# B&R Automation Studio project Lab2_Conveyor (part 3)

#### StateMoveToMagazine.ld
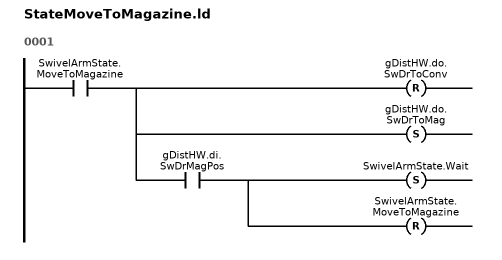
Ladder, written as Structured Text:
```iecst
ACTION StateMoveToMagazine:
VAR
    _p1 : BOOL;
END_VAR
(* Network 1 *)
IF SwivelArmState.MoveToMagazine THEN
    gDistHW.do.SwDrToConv := FALSE;
    gDistHW.do.SwDrToMag := TRUE;
END_IF;
_p1 := SwivelArmState.MoveToMagazine AND gDistHW.di.SwDrMagPos;
IF _p1 THEN
    SwivelArmState.Wait := TRUE;
    SwivelArmState.MoveToMagazine := FALSE;
END_IF;
END_ACTION
```

### Program Logical/Distributing/AlarmCtrl (IEC) - Alarm control for distributor

#### Cyclic.ld - Cyclic code
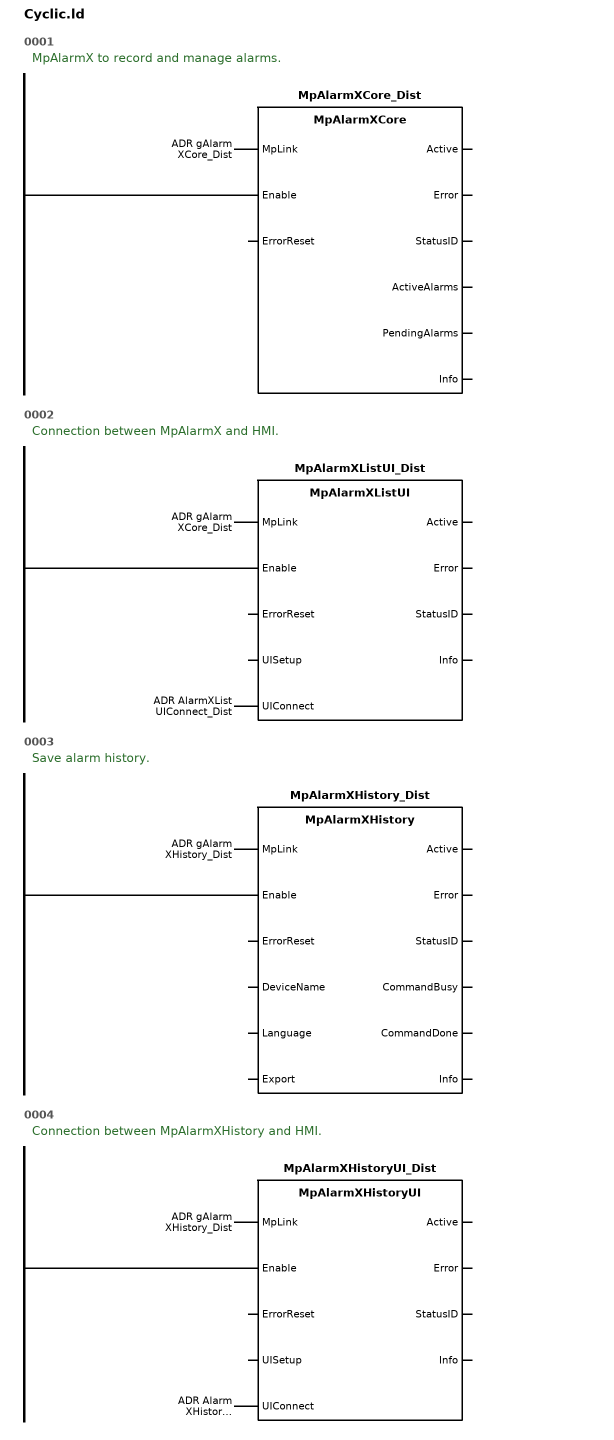
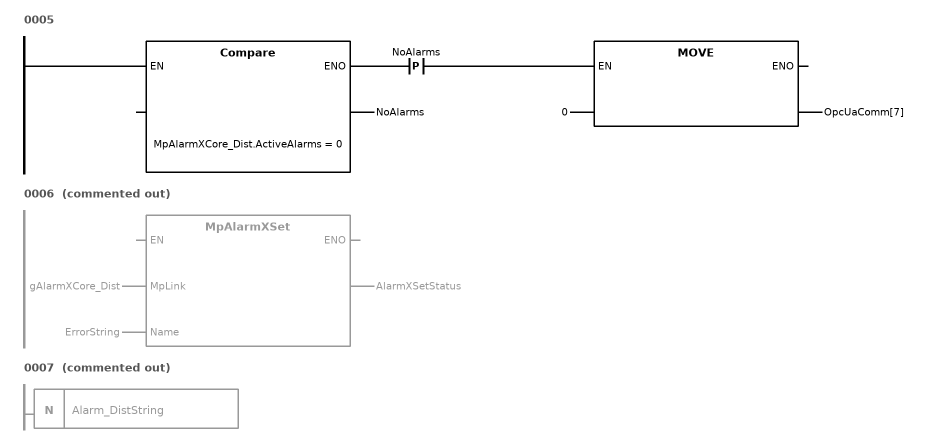
Ladder, written as Structured Text:
```iecst
(*********************************************************************************
 * Copyright: 	Hartfiel Automation
 * Author:    	cashley
 * Created:   	March 8, 2019/12:40 PM
 * Description: 	This file contains alarm handling for the distributing 			station.
 *********************************************************************************)
PROGRAM _CYCLIC
VAR
    _e1 : R_TRIG;
END_VAR
(* Network 1: MpAlarmX to record and manage alarms. *)
MpAlarmXCore_Dist(MpLink := ADR(gAlarmXCore_Dist), Enable := TRUE);

(* Network 2: Connection between MpAlarmX and HMI. *)
MpAlarmXListUI_Dist(MpLink := ADR(gAlarmXCore_Dist), Enable := TRUE, UIConnect := ADR(AlarmXListUIConnect_Dist));

(* Network 3: Save alarm history. *)
MpAlarmXHistory_Dist(MpLink := ADR(gAlarmXHistory_Dist), Enable := TRUE);

(* Network 4: Connection between MpAlarmXHistory and HMI. *)
MpAlarmXHistoryUI_Dist(MpLink := ADR(gAlarmXHistory_Dist), Enable := TRUE, UIConnect := ADR(AlarmXHistoryUIConnect_Dist));

(* Network 5 *)
NoAlarms := MpAlarmXCore_Dist.ActiveAlarms = 0;
_e1(CLK := NoAlarms);
IF _e1.Q THEN OpcUaComm[7] := 0; END_IF;

(* Network 6 *) (* commented out *)
// AlarmXSetStatus := MpAlarmXSet(MpLink := gAlarmXCore_Dist, Name := ErrorString);

(* Network 7 *) (* commented out *)
// Alarm_DistString;
END_PROGRAM
```

#### Variables.var - Local variables
```iecst
VAR
	MpAlarmXCore_Dist : MpAlarmXCore; (*Funciton block for MpAlarmXCore*)
	MpAlarmXListUI_Dist : MpAlarmXListUI; (*Function block for MpAlarmXListUI*)
	AlarmXListUIConnect_Dist : MpAlarmXListUIConnectType; (*MpAlarmXListUIConnect type*)
	MpAlarmXHistory_Dist : MpAlarmXHistory; (*Function block for MpAlarmXHistory*)
	MpAlarmXHistoryUI_Dist : MpAlarmXHistoryUI; (*Function block for MpAlarmXHistoryUI*)
	AlarmXHistoryUIConnect_Dist : MpAlarmXHistoryUIConnectType; (*MpAlarmXHistoryUIConnect type*)
	ErrorString : STRING[255]; (*String for MpAlarmXSet*)
	AlarmXSetStatus : UDINT; (*Output status for AlarmXSet*)
	NoAlarms : BOOL;
END_VAR
```

#### Alarm_DistString.st - Alarm action file
```iecst
ACTION Alarm_DistString:

END_ACTION
```

### DistMain.typ - Package global types
```iecst
TYPE
	AutoManualSelector_Enum :
		( (*Enumeration of manual-automatic mode*)
		DISTCTRL_AUTO := 0,
		DISTCTRL_MANUAL := 1
		);
	MainCtrlRejectionCode_Enum :
		( (*Enumeration of rejection codes thrown in response to a user requesting an illegal manual action.*)
		DIST_IN_AUTO_MODE := 0, (*Rejection Code thrown when any manual command is issued while the machine is in automatic mode.*)
		EJECTOR_EXTEND_PUCK_IN_TRAY := 1, (*Rejection Code thrown when an ejector extension is requested with a puck already in the ejector tray.*)
		EJECTOR_EXTEND_SWIVEL_IN_TRAY := 2, (*Rejection Code thrown when an ejector is requested with the swivel arm in the magazine position.*)
		SWIVEL_MOVE_MAG_HOLDING_PUCK := 3, (*Rejection Code thrown when the user tries to move the swivel arm to the magazine while the arm is holding a puck. Prevents pucks from being moved back to the ejector station, once removed.*)
		SWIVEL_MOVE_CONV_PUCK_CONFLICT := 4, (*Rejection Code thrown when the user attempts to transfer a puck to the conveyor with a puck already at the conveyor start position.*)
		SWIVEL_VAC_ON_NO_PRODUCT := 5, (*Rejection Code thrown when the user attempts to activate the swivel arm vacuum when there is no product under the suction cup.*)
		SWIVEL_VAC_OFF_PUCK_IN_TRANSIT := 6, (*Rejection Code thrown when the user attempts to deactivate the swivel arm vacuum while a puck is held and the swivel arm is in an intermediate position.*)
		CONV_JOG_BACK_PUCK_AT_START := 7, (*Rejection Code thrown when the user attempts to jog the conveyor backwards such that a puck falls off the conveyor.*)
		DIST_REJECT_PLACEHOLDER := 999,
		EJECTOR_EXTEND_ALREADY_IN_POS := 8, (*Rejection Code thrown when the user attempts to extend the ejection cylinder when it is already in the extended position.*)
		EJECTOR_RETRACT_ALREADY_IN_POS := 9, (*Rejection Code thrown when the user attempts to retract the ejection cylinder when it is already in the retracted position.*)
		SWIVEL_TO_MAG_ALREADY_IN_POS := 10, (*Rejection Code thrown when the user attempts to move the Swivel Arm to the magazine while to Swivel arm is already in that position.*)
		SWIVEL_TO_CONV_ALREADY_IN_POS := 11 (*Rejection Code thrown when the user attempts to move the Swivel Arm to the conveyor while to Swivel arm is already in that position.*)
		);
	MainCtrl_typ : 	STRUCT  (*Top-level interface structure for the MainCtrl task*)
		Input : MainCtrlInput_typ;
		Output : MainCtrlOutput_typ;
	END_STRUCT;
	MainCtrlInput_typ : 	STRUCT  (*Contains command and parameter substructures for the MainCtrl interface*)
		Cmd : MainCtrlCmd_typ; (*Command for MainCtrl*)
		Par : MainCtrlPar_typ; (*Parameters for MainCtrl*)
	END_STRUCT;
	MainCtrlCmd_typ : 	STRUCT  (*Contains commands for the MainCtrl interface*)
		StartAuto : BOOL;
		StopAuto : BOOL;
		Home : BOOL;
		Ejector : MainCtrlCmdEjector_typ; (*Contains a command substructure for the Ejector station*)
		SwivelArm : MainCtrlCmdSwivelArm_typ; (*Contains a command substructure for the Swivel Arm station*)
		Conveyor : MainCtrlCmdConveyor_typ; (*Contains a command substructure for the Conveyor station*)
		Reset : BOOL;
	END_STRUCT;
	MainCtrlCmdEjector_typ : 	STRUCT  (*Contains commands for the Ejector station*)
		Extend : BOOL; (*Command to extend the Ejector cylinder*)
		Retract : BOOL; (*Command to retract the Ejector cylinder*)
	END_STRUCT;
	MainCtrlCmdSwivelArm_typ : 	STRUCT  (*Contains commands for the Swivel Arm station*)
		MoveToConveyor : BOOL; (*Command to move the Swivel Arm to the Conveyor position*)
		MoveToMagazine : BOOL; (*Command to move the Swivel Arm to the magazine (i.e. Ejector) position*)
		VacuumOnImpulse : BOOL; (*Command to activate the Swivel Arm vacuum for an impulse. Used to pick up products.*)
		VacuumOffImpulse : BOOL; (*Command to active the Swivel Arm vacuum ejection impulse. Used to drop products.*)
	END_STRUCT;
	MainCtrlCmdConveyor_typ : 	STRUCT  (*Contains commands for the Conveyor station*)
		JogFwd : BOOL; (*Command to jog the Conveyor forward.*)
		JogBack : BOOL; (*Command to jog the Conveyor backward.*)
	END_STRUCT;
	MainCtrlPar_typ : 	STRUCT  (*Contains parameters for the MainCtrl task*)
		Mode : AutoManualSelector_Enum; (*Parameter to select manual/automatic operation.*)
		Conveyor : MainCtrlParConveyor_typ; (*Contains parameters for the Conveyor station*)
	END_STRUCT;
	MainCtrlParConveyor_typ : 	STRUCT  (*Contains parameters for the Conveyor station*)
		Speed : REAL; (*Parameter to set the speed of the conveyor. This value is applied to the Jog Forward, Jog Backward, and MoveVelocity actions for the conveyor.*)
		Accel : REAL; (*Parameter to set the acceleration of the conveyor. This value is applied to the Jog Forward, Jog Backward, and MoveVelocity actions for the conveyor.*)
		Decel : REAL; (*Parameter to set the deceleration of the conveyor. This value is applied to the Jog Forward, Jog Backward, and MoveVelocity actions for the conveyor.*)
	END_STRUCT;
	MainCtrlOutput_typ : 	STRUCT  (*Contains Status and "Command Rejected" information related to the MainCtrl task*)
		CommandRejected : BOOL; (*Output to indicate that a requested command is not allowed at a given time. True if the command is forbidden, false otherwise.*)
		RejectionCode : MainCtrlRejectionCode_Enum; (*Provides more detailed information about which command was rejected, and why.*)
		Status : MainCtrlStatus_typ; (*Provides additional status information about the MainCtrl task.*)
	END_STRUCT;
	MainCtrlStatus_typ : 	STRUCT  (*Contains status information about the MainCtrl task*)
		AutoRunTime : TIME; (*Time the machine has continuously been in automatic mode.*)
		DistProductCount : UDINT; (*Counter for how many products have been distributed by the distribution side of the machine.*)
		IsHomed : BOOL; (*Indicates whether the distribution half of the machine has been homed. True of the machine is homed.*)
	END_STRUCT;
END_TYPE
```

### DistMain.var - Package global variables
```iecst
VAR
	OpcUaComm : ARRAY[0..7] OF USINT; (*Communcation structure for OPCUA*)
	MainCtrl : MainCtrl_typ := (Input:=(Par:=(Mode:=DISTCTRL_MANUAL,Conveyor:=(Speed:=15.0,Accel:=200.0,Decel:=200.0)))); (*MainCtrl interface structure*)
END_VAR
```

### Program Logical/Distributing/dummyprog

#### Variables.var
```iecst
VAR
	ButtonLocked : ARRAY[0..2,0..2] OF BOOL := [FALSE,2(TRUE),FALSE,2(TRUE),FALSE,2(TRUE)];
	ButtonPressed : ARRAY[0..2,0..2] OF BOOL := [TRUE,2(FALSE),TRUE,2(FALSE),TRUE,2(FALSE)];
	i : USINT := 0;
	colourassigned : BOOL := FALSE;
	Lane : USINT := 0;
	Colour : USINT := 0;
END_VAR
VAR CONSTANT
	NUMBER_OF_LANES : USINT := 3;
	NUMBER_OF_COLOURS : USINT := 3;
	MAI_LANES : USINT := NUMBER_OF_LANES - 1;
	MAI_COLOURS : USINT := NUMBER_OF_COLOURS - 1;
END_VAR
VAR
	RTRIG : ARRAY[0..2,0..2] OF R_TRIG;
END_VAR
```

#### Cyclic.st
```iecst
PROGRAM _CYCLIC
	FOR Colour := 0 TO MAI_COLOURS BY 1 DO
		FOR Lane := 0 TO MAI_LANES BY 1 DO
			RTRIG[Colour,Lane].CLK := ButtonPressed[Colour,Lane];
		END_FOR
	END_FOR

	FOR Colour := 0 TO MAI_COLOURS BY 1 DO
		colourassigned := FALSE;
		FOR Lane := 0 TO MAI_LANES BY 1 DO
			IF ButtonPressed[Colour,Lane] THEN
				colourassigned := TRUE;
				FOR i := 0 TO MAI_LANES BY 1 DO
					IF i <> Lane THEN
						ButtonLocked[Colour,i] := TRUE;
					END_IF
				END_FOR
			END_IF
		END_FOR

		IF colourassigned = FALSE THEN
			FOR Lane := 0 TO MAI_LANES BY 1 DO
				ButtonLocked[Colour,Lane] := FALSE;
			END_FOR
		END_IF
	END_FOR

	FOR Lane := 0 TO MAI_LANES BY 1 DO
		FOR Colour := 0 TO MAI_COLOURS BY 1 DO
			IF RTRIG[Colour,Lane].Q THEN
				FOR i := 0 TO MAI_COLOURS BY 1 DO
					ButtonPressed[i,Lane] := FALSE;
				END_FOR
			END_IF
		END_FOR
	END_FOR

	FOR Colour := 0 TO MAI_COLOURS BY 1 DO
		FOR Lane := 0 TO MAI_LANES BY 1 DO
			RTRIG[Colour,Lane]();
		END_FOR
	END_FOR

END_PROGRAM
```

### Package Logical/Sorting - Sorter configuration

### Package Logical/Sorting/gAxisSortobj - gAxisSortobj

### Data object Logical/Sorting/gAxisSortobj/gAxisSorta (Apt) - gAxisSorta

#### gAxisSorta.apt
```
AcoposParameterTable:
  Root Parameters:
    64232 = 51200 (Name=SM_SCALE_STEP)
    64233 = 1000 (Name=SM_SCALE_LOAD_UNITS)
    64234 = 1 (Name=SM_SCALE_LOAD_MOTREV)
    230 = PCTRL_S_SET (Name=PCTRL_S_ACT_PARID)  // CTRL Position controller: Actual encoder position parameter ID
```

- Data object Logical/Sorting/gAxisSortobj/gAxisSorti (Ax) - gAxisSorti (no source held here)

### SortGlobal.var - Package global variables
```iecst
VAR
	gSortHW : gSortHW_type; (*Control variable for hardware IO types for sorter*)
	MpAlarmXCore_Sort : MpAlarmXCore; (*Function block for MpAlarmXCore*)
	MpAlarmXListUI_Sort : MpAlarmXListUI; (*Function block for MpAlarmXListUI*)
	AlarmXListUIConnect_Sort : MpAlarmXListUIConnectType; (*MpAlarmXListUIConnect type*)
	MpAlarmXHistory_Sort : MpAlarmXHistory; (*Function block for MpAlarmXHistory*)
	MpAlarmXHistoryUI_Sort : MpAlarmXHistoryUI; (*Function block for MpAlarmXHistoryUI*)
	AlarmXHistoryUIConnect_Sort : MpAlarmXHistoryUIConnectType; (*MpAlarmXHistoryUIConnect type*)
	gSortModuleOK : gSortModuleOK_type; (*Control variable for sorter module statuses*)
	ErrorString : STRING[255]; (*String for MpAlarmXSet unique alarm code*)
	AlarmXSetStatus : UDINT; (*Output status for AlarmXSet*)
END_VAR
```

### SortGlobal.typ - Package global types
```iecst
TYPE
	gSortHW_type : 	STRUCT  (*Hardware IO types for sorter*)
		di : diSort_type; (*Digital inputs for sorter*)
		do : doSort_type; (*Digital outputs for sorter*)
	END_STRUCT;
	diSort_type : 	STRUCT  (*Digital inputs for sorter*)
		ProductAvailable : BOOL; (*Product available*)
		Metallic : BOOL; (*Metallic product*)
		NotBlack : BOOL; (*Product is not black*)
		LaneFull : BOOL; (*Lane full*)
		Switch1Retracted : BOOL; (*Switch 1 retracted*)
		Switch1Extended : BOOL; (*Switch 1 extended*)
		Switch2Retracted : BOOL; (*Switch 2 retracted*)
		Switch2Extended : BOOL; (*Switch 2 extended*)
	END_STRUCT;
	doSort_type : 	STRUCT  (*Digital outputs for sorter*)
		ExtendSwitch1 : BOOL; (*Extend switch 1*)
		ExtendSwitch2 : BOOL; (*Extend switch 2*)
		RetractStopper : BOOL; (*Retract stopper*)
	END_STRUCT;
	gSortModuleOK_type : 	STRUCT  (*Sorter module statuses*)
		Interface : BOOL; (*5PP5IF.FPLM-00 status*)
		BusController : BOOL; (*X20BC0083 status*)
		PowerSupply : BOOL; (*X20PS9400 status*)
		DigitalInput : BOOL; (*X20DI9371 status*)
		PotentialDist0012 : BOOL; (*X20PD0012 status*)
		PotentialDist0011 : BOOL; (*X20PD0011 status*)
		DigitalOutput : BOOL; (*X20DO9322 status*)
		BusTransmitter : BOOL; (*X20BT9100 status*)
		StepperMotor : BOOL; (*X67SM2436 status*)
	END_STRUCT;
END_TYPE
```

### Station.typ - Local data types
```iecst
TYPE
	CMD_type : 	STRUCT  (*Station command type*)
		RetractStopper : BOOL; (*Retract stopper*)
		ExtendSwitch1 : BOOL; (*Extend switch 1*)
		ExtendSwitch2 : BOOL; (*Extend switch 2*)
		RunCycle : BOOL; (*Run cycle*)
		ErrorReset : BOOL; (*Reset error*)
		Home : BOOL; (*Home machine*)
	END_STRUCT;
	Color_enum :
		( (*Color selector enumeration*)
		NONE := 0, (*No color*)
		RED := 1, (*Red color*)
		BLACK := 2, (*Black color*)
		METALLIC := 3 (*Metallic color*)
		);
	Conveyor_type : 	STRUCT  (*Conveyor type for motion control*)
		MoveAdditive : BOOL; (*Move additive for conveyor*)
		MoveVelocity : BOOL; (*Move velocity for conveyor*)
		Stop : BOOL; (*Stop conveyor*)
		Velocity : REAL; (*Conveyor velocity parameter*)
		Accel : REAL; (*Conveyor acceleration parameter*)
		Decel : REAL; (*Conveyor deceleration parameter*)
		JogPos : BOOL; (*Jog conveyor forward*)
		JogNeg : BOOL; (*Jog conveyor backward*)
		Home : BOOL; (*Home the conveyor*)
		MoveActive : BOOL; (*Conveyor move active*)
		InPosition : BOOL; (*Conveyor in position*)
		Ready : BOOL; (*Conveyor ready*)
	END_STRUCT;
	Index_enum :
		( (*Index enumeration for sorting station*)
		AUTO := 0, (*Auto index*)
		ISSUED := 1, (*Issued index*)
		ERROR := 2, (*Error index*)
		DISPENSER := 3, (*Dispenser index*)
		FLIPPER := 4, (*Flipper index*)
		CONVEYOR := 5, (*Conveyor index*)
		SORTER := 6, (*Sorter index*)
		COLLECTOR := 7 (*Collector index*)
		);
	Input_type : 	STRUCT  (*Input type for sorting station*)
		CMD : CMD_type; (*Command type*)
		Par : Par_type; (*Parameter type*)
	END_STRUCT;
	Output_type : 	STRUCT  (*Output type for sorting station*)
		Status : Status_type; (*Status type*)
		Time : UDINT; (*Automatic mode run time*)
		CommandRejected : BOOL; (*Command has been rejected*)
		RejectionCode : UDINT; (*Rejection code*)
	END_STRUCT;
	Par_type : 	STRUCT  (*Parameters type for lane selection*)
		ParID : ARRAY[0..2]OF Color_enum := [RED,BLACK,METALLIC]; (*Array for Sorting order, Index 0 (Left Slide) - 2 (Right Slide)  Color Corresponding to Station*)
	END_STRUCT;
	SlotIndex_type : 	STRUCT  (*Lane selector index type*)
		Left : USINT; (*Lane 1 slot*)
		Middle : USINT; (*Lane 2 slot*)
		Right : USINT; (*Lane 3 slot*)
	END_STRUCT;
	Slot_type : 	STRUCT  (*Lane selector slot type*)
		Left : Color_enum; (*Lane 1 slot*)
		Middle : Color_enum; (*Lane 2 slot*)
		Right : Color_enum; (*Lane 3 slot*)
	END_STRUCT;
	Station_type : 	STRUCT  (*Station type for sorting station*)
		Output : Output_type; (*Output type*)
		Input : Input_type; (*Input type*)
		ColorCount : ARRAY[0..2]OF USINT; (*Puck Color Count [Red, Black, Metallic]*)
		Reset : BOOL;
		Conveyor : Conveyor_type; (*Conveyor type*)
		OpcUa : OpcUa_type; (*OpcUa type*)

	END_STRUCT;
	Status_type : 	STRUCT  (*Status type for sorting station*)
		Switch1Extended : BOOL; (*Switch 1 extended*)
		Switch1Retracted : BOOL; (*Switch 1 retracted*)
		Switch2Extended : BOOL; (*Switch 2 extended*)
		Switch2Retracted : BOOL; (*Switch 2 retracted*)
		Error : BOOL; (*Error has been detected*)
		ErrorID : UDINT; (*Error ID*)
		IsHomed : BOOL; (*Sorting station is homed*)
		ProductAvailable : BOOL; (*Product available*)
		MetallicProduct : BOOL; (*Metallic product*)
		LaneFull : BOOL; (*Lane is full*)
		ProductNotBlack : BOOL; (*Product not black*)
		SlotFull : ARRAY[0..2]OF BOOL; (*Slot is full*)
		Occupied : BOOL; (*Occupied*)
	END_STRUCT;
	OpcUa_type : 	STRUCT  (*OpcUa type for server connection*)
		Write : BOOL; (*Write OPCUA*)
		Read : BOOL; (*Read OPCUA*)
		Connect : BOOL; (*Connect to OPCUA*)
		Disconnect : BOOL; (*Disconnect to OPCUA*)
	END_STRUCT;
END_TYPE
```

### Station.var - Local variables
```iecst
VAR
	Station : Station_type; (*Station type*)
	OpcUaComm : ARRAY[0..7] OF USINT; (*OpcUa variable*)
	OpcUaCommOld : ARRAY[0..7] OF USINT; (*OpcUa old variable*)
	OpcUaCommTemp : ARRAY[0..7] OF USINT; (*OpcUa temp variable*)
	MachineState : ARRAY[0..7] OF USINT; (*Machine state variable*)
	MachineStateOld : ARRAY[0..7] OF USINT; (*Machine state old variable*)
	MachineStateTemp : ARRAY[0..7] OF USINT; (*Machine state temp variable*)
END_VAR
```

- Visualisation Logical/Sorting/Visualization (not shown)

### Package Logical/Sorting/OPCUA - OPCUA package

### Program Logical/Sorting/OPCUA/OPCUAClient (IEC) - OPCUA Client

#### Types.typ
```iecst
TYPE
	ClientState_enum :
		( (*State enumeration for OPCUA client*)
		CLIENT_INIT, (*Initialize and execute connect command*)
		CLIENT_CONNECT, (*Client connecting to server*)
		CLIENT_GET_NS, (*Getting namespace*)
		CLIENT_CHECK_NS, (*Check for namespace error*)
		CLIENT_GET_NH, (*Getting node handle*)
		CLIENT_CHECK_NH, (*Check for node handle error*)
		CLIENT_IDLE, (*Client idle*)
		CLIENT_READ, (*Read item*)
		CLIENT_CHECK_READ, (*Check for read error*)
		CLIENT_WRITE, (*Write to item*)
		CLIENT_CHECK_WRITE, (*Check for write error*)
		CLIENT_NH_RELEASE, (*Release node handle*)
		CLIENT_CHECK_RELEASE, (*Check for node handle release error*)
		CLIENT_DISCONNECT, (*Client disconnecting from server*)
		CLIENT_CHECK_DISCONNECT, (*Check for disconnect error*)
		CLIENT_ERROR (*An error has been detected*)
		);
END_TYPE
```

#### Variables.var
```iecst
VAR
	UAConnected : BOOL; (*Connection is established between client and server*)
	ClientState : ClientState_enum; (*State of OPCUA client*)
END_VAR
```

#### Cyclic.st
```iecst
(*********************************************************************************
 * Copyright: 	Hartfiel Automation
 * Author:    	cashley
 * Created:   	March 8, 2019/12:40 PM
 * Description: This file contains a state machine for the client that details
				the process of establishing a client connection to the OPCUA server.
 *********************************************************************************)
PROGRAM _CYCLIC

	CASE ClientState OF

		CLIENT_INIT: //Initialize and execute connection
			ExecuteConnect := TRUE;
			ClientState    := CLIENT_CONNECT;

		CLIENT_CONNECT: //Establish connection to OPCUA server and check for error
			IF EDGEPOS(UaConnect_0.Done) THEN
				IF NOT UaConnect_0.Error THEN //Check for error
					ClientState := CLIENT_GET_NS;
					UAConnected := TRUE;
				ELSE
					ClientState := CLIENT_ERROR;
				END_IF
				ExecuteConnect  := FALSE;
			END_IF

		CLIENT_GET_NS: //Get namespace index
			ExecuteGetnamespaceIndex := TRUE;
			ClientState 			 := CLIENT_CHECK_NS;

		CLIENT_CHECK_NS: //Read index of required namespace for PVs and check for error
			IF EDGEPOS(UaGetNamespaceIndex_0.Done) THEN
				IF NOT UaGetNamespaceIndex_0.Error THEN
					ClientState := CLIENT_GET_NH;
				ELSE
					ClientState := CLIENT_ERROR;
				END_IF
				ExecuteGetnamespaceIndex := FALSE;
			END_IF

		CLIENT_GET_NH: //Get node handle
			ExecuteNodeGetHandle := TRUE;
			ClientState 		 := CLIENT_CHECK_NH;

		CLIENT_CHECK_NH: //Get handle for required node and check for error
			IF EDGEPOS(UaNodeGetHandle_0.Done) THEN
				IF NOT UaNodeGetHandle_0.Error THEN
					ClientState 		  := CLIENT_IDLE;
					Station.OpcUa.Connect := FALSE;
				ELSE
					ClientState := CLIENT_ERROR;
				END_IF
				ExecuteNodeGetHandle := FALSE;
			END_IF

		CLIENT_IDLE: //Idle - waiting for command to read, write, disconnect, or reconnect
			IF Station.OpcUa.Connect = TRUE THEN
				ClientState 		  := CLIENT_INIT;
				Station.OpcUa.Connect := FALSE;
			ELSIF Station.OpcUa.Disconnect THEN
				ClientState 			 := CLIENT_NH_RELEASE;
				Station.OpcUa.Disconnect := FALSE;
			ELSIF Station.OpcUa.Read AND UAConnected THEN
				ClientState := CLIENT_READ;
			ELSIF Station.OpcUa.Write AND UAConnected THEN
				ClientState := CLIENT_WRITE;
			END_IF

		CLIENT_READ: //Read plc variable from server
			ExecuteRead := TRUE;
			ClientState := CLIENT_CHECK_READ;

		CLIENT_CHECK_READ: //Read variable from OPCUA Server and check for error
			IF EDGEPOS(UaRead_0.Done) THEN
				IF NOT UaRead_0.Error THEN
					ClientState := CLIENT_IDLE;
				ELSE
					ClientState := CLIENT_ERROR;
				END_IF
				ExecuteRead 	   := FALSE;
				Station.OpcUa.Read := FALSE;
			END_IF

		CLIENT_WRITE: //Write plc variable to server
			ExecuteWrite := TRUE;
			ClientState  := CLIENT_CHECK_WRITE;

		CLIENT_CHECK_WRITE: //Write variable to required node from OPCUA Server and check for error
			IF EDGEPOS(UaWrite_0.Done) THEN
				IF NOT UaWrite_0.Error THEN
					ClientState := CLIENT_IDLE;
				ELSE
					ClientState := CLIENT_ERROR;
				END_IF
				ExecuteWrite 	    := FALSE;
				Station.OpcUa.Write := FALSE;
			END_IF

		CLIENT_NH_RELEASE: //Release node handle
			ExecuteNodeReleaseHandle := TRUE;
			ClientState 		 	 := CLIENT_CHECK_RELEASE;

		CLIENT_CHECK_RELEASE: //Release handle for node and check for error
			IF EDGEPOS(UaNodeReleaseHandle_0.Done) THEN
				IF NOT UaNodeReleaseHandle_0.Error THEN
					ClientState := CLIENT_DISCONNECT;
				ELSE
					ClientState := CLIENT_ERROR;
				END_IF
				ExecuteNodeReleaseHandle := FALSE;
			END_IF

		CLIENT_DISCONNECT: //Disconnect from OPCUA server
			ExecuteDisconnect := TRUE;
			ClientState    	  := CLIENT_CHECK_DISCONNECT;

		CLIENT_CHECK_DISCONNECT: //Disconnect from OPCUA server and check for error
			IF EDGEPOS(UaDisconnect_0.Done) THEN
				IF NOT UaDisconnect_0.Error THEN
					ClientState := CLIENT_IDLE;
					UAConnected := FALSE;
				ELSE
					ClientState := CLIENT_ERROR;
				END_IF
				Station.OpcUa.Disconnect := FALSE;
				ExecuteDisconnect 		 := FALSE;
			END_IF

		CLIENT_ERROR: //An error has been detected
			ExecuteConnect  		 := FALSE;
			ExecuteGetnamespaceIndex := FALSE;
			ExecuteNodeGetHandle     := FALSE;
			ExecuteRead 			 := FALSE;
			ExecuteWrite 			 := FALSE;
			ExecuteNodeReleaseHandle := FALSE;
			ExecuteDisconnect 		 := FALSE;
			ClientState 			 := CLIENT_IDLE;

	END_CASE

END_PROGRAM
```

#### Init.st
```iecst
PROGRAM _INIT

END_PROGRAM
```

### Program Logical/Sorting/OPCUA/OPCUAConnect (IEC) - OPCUA Connection

#### Cyclic.st
```iecst
(*********************************************************************************
 * Copyright: 	Hartfiel Automation
 * Author:    	cashley
 * Created:   	March 9, 2019/12:02 PM
 * Description: This file contains the function blocks and parameters for the
				process of establishing a client connection to the OPCUA server.
 *********************************************************************************)
PROGRAM _CYCLIC

	//Session connect information - connection to OPCUA server
	UaSessionConnectInfo.SecurityMsgMode 						 := UASecurityMsgMode_None;
	UaSessionConnectInfo.SecurityPolicy 						 := UASecurityPolicy_None;
	UaSessionConnectInfo.TransportProfile 					   	 := UATP_UATcp;
	UaSessionConnectInfo.UserIdentityToken.UserIdentityTokenType := UAUITT_Anonymous;
	UaSessionConnectInfo.SessionTimeout 						 := SESSION_TIMEOUT;
	UaSessionConnectInfo.MonitorConnection 					   	 := MONITOR_CONNECT_TIME;

	//UaConnect - establish connection to OPCUA server
	UaConnect_0.Execute 		   := ExecuteConnect;
	UaConnect_0.ServerEndpointUrl  := SERVER_URL;
	UaConnect_0.SessionConnectInfo := UaSessionConnectInfo;
	UaConnect_0.Timeout 		   := CONNECT_INFO_TIMEOUT;

	//Check for error and determine connection handle
	IF UaConnect_0.Busy = FALSE THEN
		IF UaConnect_0.Done = TRUE THEN
			ErrorID 	  := 0;
			ConnectionHdl := UaConnect_0.ConnectionHdl;
		END_IF
		IF UaConnect_0.Error = TRUE THEN
			ErrorID 	  := UaConnect_0.ErrorID;
			ConnectionHdl := 0;
		END_IF
	END_IF

	//UaGetNamespaceIndex - read index of namespace for PVs
	UaGetNamespaceIndex_0.Execute 	  	:= ExecuteGetnamespaceIndex;
	UaGetNamespaceIndex_0.ConnectionHdl := ConnectionHdl;
	UaGetNamespaceIndex_0.NamespaceUri  := NS_URI;
	UaGetNamespaceIndex_0.Timeout 	  	:= NS_TIMEOUT;

	//Check for error and determine namespace index
	IF UaGetNamespaceIndex_0.Busy = FALSE THEN
		IF UaGetNamespaceIndex_0.Done = TRUE THEN
			ErrorID 	   := 0;
			NamespaceIndex := UaGetNamespaceIndex_0.NamespaceIndex;
		END_IF
		IF UaGetNamespaceIndex_0.Error = TRUE THEN
			ErrorID 	   := UaGetNamespaceIndex_0.ErrorID;
			NamespaceIndex := 0;
		END_IF
	END_IF

	//Node identifier information
	UaNodeID.NamespaceIndex := NamespaceIndex;
	UaNodeID.Identifier 	:= NODE_IDENTIFIER;
	UaNodeID.IdentifierType := UAIdentifierType_String;

	//UaNodeGetHandle - get handle for required node
	UaNodeGetHandle_0.Execute 	  	:= ExecuteNodeGetHandle;
	UaNodeGetHandle_0.ConnectionHdl := ConnectionHdl;
	UaNodeGetHandle_0.NodeID 		:= UaNodeID;
	UaNodeGetHandle_0.Timeout 	  	:= NH_TIMEOUT;

	//Check for error and determine node handle
	IF UaNodeGetHandle_0.Busy = FALSE THEN
		IF UaNodeGetHandle_0.Done = TRUE THEN
			ErrorID := 0;
			NodeHdl := UaNodeGetHandle_0.NodeHdl;
		END_IF
		IF UaNodeGetHandle_0.Error = TRUE THEN
			ErrorID := UaNodeGetHandle_0.ErrorID;
			NodeHdl := 0;
		END_IF
	END_IF

	//Parameters for specifying the node
	UaNodeAddInfo.AttributeId 	  := UAAI_Value;
	UaNodeAddInfo.IndexRangeCount := 0;

	Variable_Rd0 := READ_VAR;

	//UaRead - read required node from OPCUA server and write it in local plc variable
	UaRead_0(Execute  := ExecuteRead,
		ConnectionHdl := ConnectionHdl,
		NodeHdl 	  := NodeHdl,
		NodeAddInfo   := UaNodeAddInfo,
		Timeout 	  := READ_TIMEOUT,
		Variable 	  := Variable_Rd0
	);

	//Check for error
	IF (UaRead_0.Busy = 0) THEN
		IF (UaRead_0.Done = 1) THEN
			ErrorID := 0;
		END_IF
		IF (UaRead_0.Error = 1) THEN
			ErrorID := UaRead_0.ErrorID;
		END_IF
	END_IF

	//Parameters for specifying the node
	UaNodeAddInfo.AttributeId 	  := UAAI_Value;
	UaNodeAddInfo.IndexRangeCount := 0;

	Variable_Wr0 := WRITE_VAR;

	//UaWrite - write variable to required node from OPCUA server
	UaWrite_0(
		Execute 	  := ExecuteWrite,
		ConnectionHdl := ConnectionHdl,
		NodeHdl 	  := NodeHdl,
		NodeAddInfo   := UaNodeAddInfo,
		Timeout 	  := WRITE_TIMEOUT,
		Variable 	  := Variable_Wr0
		);

	//Check for error
	IF UaWrite_0.Busy = FALSE THEN
		IF UaWrite_0.Done = TRUE THEN
			ErrorID  := 0;
		END_IF
		IF UaWrite_0.Error = TRUE THEN
			ErrorID := UaWrite_0.ErrorID;
		END_IF
	END_IF

	//UaNodeReleaseHandle - release the handle for the node
	UaNodeReleaseHandle_0.Execute 	    := ExecuteNodeReleaseHandle;
	UaNodeReleaseHandle_0.ConnectionHdl := ConnectionHdl;
	UaNodeReleaseHandle_0.NodeHdl 		:= NodeHdl;
	UaNodeReleaseHandle_0.Timeout 		:= NH_RELEASE_TIMEOUT;

	//Check for error and set node handle
	IF (UaNodeReleaseHandle_0.Busy = 0) THEN
		IF (UaNodeReleaseHandle_0.Done = 1) THEN
			ErrorID := 0;
			NodeHdl := 0;
		END_IF
		IF (UaNodeReleaseHandle_0.Error = 1) THEN
			ErrorID := UaNodeReleaseHandle_0.ErrorID;
		END_IF
	END_IF

	//UaDisconnect - disconnect from OPCUA server
	UaDisconnect_0.Execute 		 := ExecuteDisconnect;
	UaDisconnect_0.ConnectionHdl := ConnectionHdl;
	UaDisconnect_0.Timeout 		 := DISCONNECT_TIMEOUT;

	//Check for error and set connection handle
	IF (UaDisconnect_0.Busy = 0) THEN
		IF ExecuteDisconnect = TRUE THEN
			ConnectionHdl := 0;
		END_IF
	END_IF

	//Call UA function blocks
	UaConnect_0();
	UaGetNamespaceIndex_0();
	UaNodeGetHandle_0();
	UaNodeReleaseHandle_0();
	UaDisconnect_0();

END_PROGRAM
```

#### Exit.st
```iecst
PROGRAM _EXIT

END_PROGRAM
```

#### Init.st
```iecst
PROGRAM _INIT

END_PROGRAM
```

### Variables.var - not listed in the package file held
```iecst
VAR
	READ_VAR : {REDUND_UNREPLICABLE} STRING[255] := '::MainCtrl:OpcUaComm'; (*Read variable*)
	WRITE_VAR : {REDUND_UNREPLICABLE} STRING[255] := '::MainCtrl:MachineState'; (*Write variable*)
	SERVER_URL : {REDUND_UNREPLICABLE} STRING[255] := 'opc.tcp://10.10.10.99:4840'; (*Server Endpoint Url*)
	NS_URI : {REDUND_UNREPLICABLE} STRING[255] := 'urn:B&R/pv/'; (*NamespaceUri*)
	NODE_IDENTIFIER : {REDUND_UNREPLICABLE} STRING[255] := '::AsGlobalPV:OpcUaComm'; (*Node identifier*)
	UaWrite_0 : UA_Write; (*Function block for UA_Write*)
	UaConnect_0 : UA_Connect; (*Function block for UA_Connect*)
	ExecuteConnect : BOOL; (*Execute connect command*)
	UaSessionConnectInfo : UASessionConnectInfo; (*Info for connect session*)
	ConnectionHdl : DWORD := 0; (*Connection handle*)
	ExecuteWrite : BOOL; (*Execute write command*)
	ErrorID : DWORD; (*ID for error*)
	UaGetNamespaceIndex_0 : UA_GetNamespaceIndex; (*Function block for UA_GetNamespaceIndex*)
	ExecuteGetnamespaceIndex : BOOL; (*Execute get namespace command*)
	NamespaceIndex : UINT := 0; (*Namespace index*)
	UaNodeGetHandle_0 : UA_NodeGetHandle; (*Function block for UA_NodeGetHandle*)
	ExecuteNodeGetHandle : BOOL; (*Execute get node handle command*)
	UaNodeID : UANodeID; (*Node identifier*)
	NodeHdl : DWORD := 0; (*Node handle*)
	UaNodeAddInfo : UANodeAdditionalInfo; (*Additional info for reading and writing*)
	Variable_0 : STRING[255]; (*OPCUA process variable*)
	UaMonitoringSettings : UAMonitoringSettings; (*Settings for monitoring*)
	MonitoredItemHdl : DWORD; (*Monitored item handle*)
END_VAR
VAR CONSTANT
	SESSION_TIMEOUT : TIME := T#1m; (*Connect session timeout*)
	MONITOR_CONNECT_TIME : TIME := T#10s; (*Monitor connection time*)
	CONNECT_INFO_TIMEOUT : TIME := T#10s; (*Session connect info timeout*)
	NS_TIMEOUT : TIME := T#5s; (*Namespace timeout*)
	NH_RELEASE_TIMEOUT : TIME := T#10s; (*Node handle release timeout*)
	NH_TIMEOUT : TIME := T#10s; (*Node handle timeout*)
END_VAR
VAR
	Variable_Wr0 : STRING[255]; (*Write to variable*)
	Variable_Rd0 : STRING[255]; (*Read variable*)
END_VAR
VAR CONSTANT
	WRITE_TIMEOUT : TIME := T#10s; (*Timeout for writing variable*)
	READ_TIMEOUT : TIME := T#10s; (*Timeout for reading variable*)
	DISCONNECT_TIMEOUT : TIME := T#10s; (*Timeout for disconnecting from server*)
END_VAR
VAR
	UaRead_0 : UA_Read; (*Function block for UA_Read*)
	ExecuteRead : BOOL; (*Execute read command*)
	UaNodeReleaseHandle_0 : UA_NodeReleaseHandle; (*Function block for UA_NodeReleaseHandle*)
	ExecuteNodeReleaseHandle : BOOL; (*Execute release node handle command*)
	UaDisconnect_0 : UA_Disconnect; (*Function block for UA_Disconnect*)
	ExecuteDisconnect : BOOL; (*Execute disconnect command*)
END_VAR
```

### Package Logical/Sorting/Machine - Sorting machine functionality

### Sort.var - Local variables
```iecst
VAR
	Sorter : Sorter_type; (*Sorter type for sorting station*)
	MpAxisBasicConveyor : MpAxisBasic; (*Function block for MpAxisBasic*)
	ConveyorParam : MpAxisBasicParType; (*MpAxisBasic parameters*)
	TP_10ms_Start : TP_10ms; (*Automatic mode timer*)
	TimeIn : UDINT; (*Time in for mode*)
	SlotIndex : USINT; (*Slot index for lane*)
	TON_10ms_Opc : TON_10ms; (*Function block for TON timer *)
	MIndex : INT; (*Machine index*)
	MchUpdate : BOOL; (*Machine update*)
END_VAR
```

### Sort.typ - Local data types
```iecst
TYPE
	Sorter_type : 	STRUCT  (*Sorter type*)
		Output : Output_type; (*Output type*)
		Input : Input_type; (*Input type*)
		Conveyor : Conveyor_type; (*Conveyor type*)
		AutoMode : BOOL; (*Automatic mode*)
		NewPuck : Color_enum; (*New product color*)
		CurrentPuck : Color_enum; (*Current product color*)
		Slot : ARRAY[0..3]OF Slot_type; (*Slot lane for product*)
		SlotIndex : SlotIndex_type; (*Slot index for product*)
		Reset : BOOL; (*Reset command for timer and counters*)
	END_STRUCT;
END_TYPE
```

### Program Logical/Sorting/Machine/MainCtrl (IEC) - Sorting main control

#### Cyclic.ld - Cyclic code
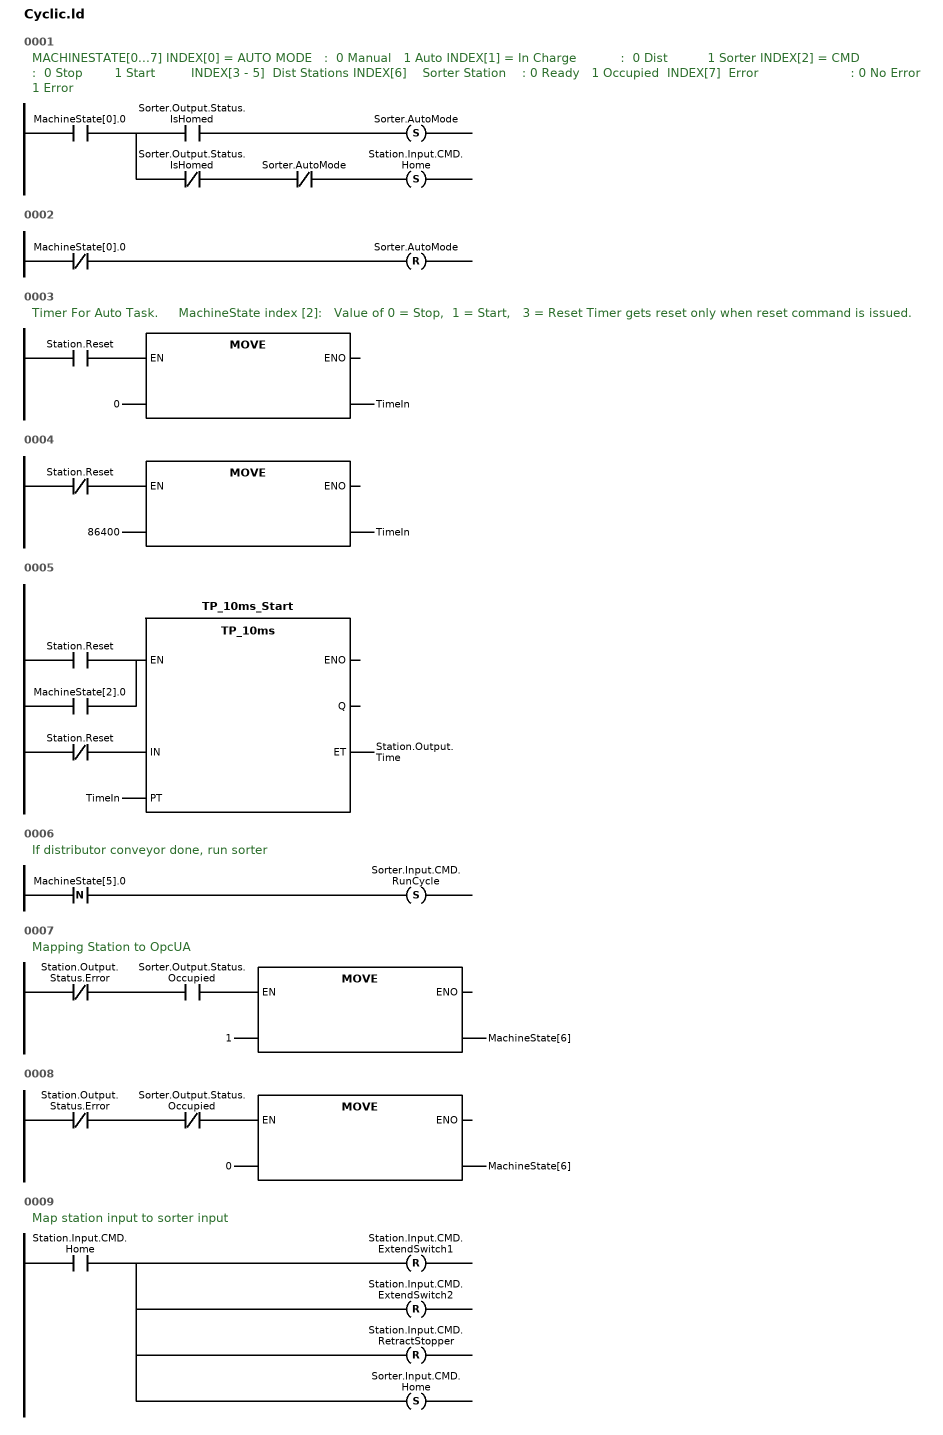
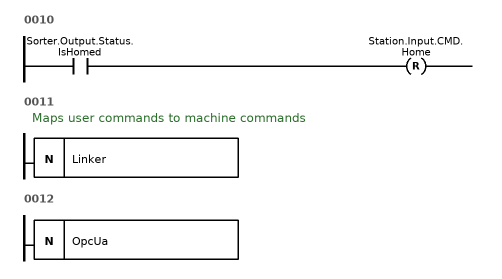
Ladder, written as Structured Text:
```iecst
(*********************************************************************************
 * Copyright: 	I-Automation
 * Author:    	John Lee
 * Created:   	March 8, 2019/12:41 PM
 * Description:   Main Ctrl task for Sorter Station
 *********************************************************************************)
PROGRAM _CYCLIC
VAR
    _e1 : F_TRIG;
    _p2 : BOOL;
END_VAR
(* Network 1: MACHINESTATE[0...7] INDEX[0] = AUTO MODE   :  0 Manual   1 Auto INDEX[1] = In Charge           :  0 Dist          1 Sorter INDEX[2] = CMD                    :  0 Stop        1 Start         INDEX[3 - 5]  Dist Stations INDEX[6]    Sorter Station    : 0 Ready   1 Occupied  INDEX[7]  Error                       : 0 No Error    1 Error  *)
IF MachineState[0].0 AND Sorter.Output.Status.IsHomed THEN Sorter.AutoMode := TRUE; END_IF;
IF MachineState[0].0 AND NOT Sorter.Output.Status.IsHomed AND NOT Sorter.AutoMode THEN
    Station.Input.CMD.Home := TRUE;
END_IF;

(* Network 2 *)
IF NOT MachineState[0].0 THEN Sorter.AutoMode := FALSE; END_IF;

(* Network 3: Timer For Auto Task.     MachineState index [2]:   Value of 0 = Stop,  1 = Start,   3 = Reset Timer gets reset only when reset command is issued.  *)
IF Station.Reset THEN TimeIn := 0; END_IF;

(* Network 4 *)
IF NOT Station.Reset THEN TimeIn := 86400; END_IF;

(* Network 5 *)
IF Station.Reset OR MachineState[2].0 THEN
    TP_10ms_Start(IN := NOT Station.Reset, PT := TimeIn);
    Station.Output.Time := TP_10ms_Start.ET;
END_IF;

(* Network 6: If distributor conveyor done, run sorter *)
_e1(CLK := MachineState[5].0);
IF _e1.Q THEN Sorter.Input.CMD.RunCycle := TRUE; END_IF;

(* Network 7: Mapping Station to OpcUA  *)
IF NOT Station.Output.Status.Error AND Sorter.Output.Status.Occupied THEN MachineState[6] := 1; END_IF;

(* Network 8 *)
IF NOT Station.Output.Status.Error AND NOT Sorter.Output.Status.Occupied THEN
    MachineState[6] := 0;
END_IF;

(* Network 9: Map station input to sorter input *)
_p2 := Station.Input.CMD.Home;
IF Station.Input.CMD.Home THEN Station.Input.CMD.ExtendSwitch1 := FALSE; END_IF;
IF _p2 THEN
    Station.Input.CMD.ExtendSwitch2 := FALSE;
    Station.Input.CMD.RetractStopper := FALSE;
    Sorter.Input.CMD.Home := TRUE;
END_IF;

(* Network 10 *)
IF Sorter.Output.Status.IsHomed THEN Station.Input.CMD.Home := FALSE; END_IF;

(* Network 11: Maps user commands to machine commands *)
Linker;

(* Network 12 *)
OpcUa;
END_PROGRAM
```

#### Init.ld - Initialization code
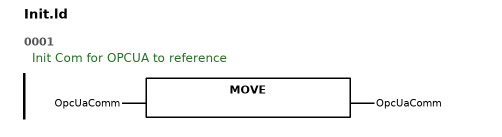
Ladder, written as Structured Text:
```iecst
PROGRAM _INIT
(* Network 1: Init Com for OPCUA to reference *)
OpcUaComm := OpcUaComm;
END_PROGRAM
```

#### Package Logical/Sorting/Machine/MainCtrl/Action - Actions

#### Linker.st
```iecst
(*********************************************************************************
 * Copyright: I-Automation
 * Author:    John Lee
 * Created:   March 15, 2019/1:19 AM
 *            Main connection point to sorter task
 *********************************************************************************)

ACTION Linker:

	// Output to Station
	Station.Output.Status.IsHomed := Sorter.Output.Status.IsHomed;
	Station.Output.Status.Switch1Extended := Sorter.Output.Status.Switch1Extended;
	Station.Output.Status.Switch1Retracted := Sorter.Output.Status.Switch1Retracted;
	Station.Output.Status.Error := Sorter.Output.Status.Error;
	Station.Output.Status.ErrorID := Sorter.Output.Status.ErrorID;
	Station.Output.RejectionCode := Sorter.Output.RejectionCode;
	Station.Output.CommandRejected := Sorter.Output.CommandRejected;
	Sorter.Reset := Station.Reset;

	// Input to Station
	Sorter.Conveyor.Velocity := Station.Conveyor.Velocity;
	Sorter.Conveyor.Accel := Station.Conveyor.Accel;
	Sorter.Conveyor.Decel := Station.Conveyor.Decel;

	//Index of Slot Array
	Station.ColorCount[0] := 0;
	Station.ColorCount[1] := 0;
	Station.ColorCount[2] := 0;

	//Counts the colors from Slot index
	FOR SlotIndex := 0 TO 3 BY 1 DO
		IF Sorter.Slot[SlotIndex].Left = RED THEN
			Station.ColorCount[0] := Station.ColorCount[0] + 1;
		END_IF
		IF Sorter.Slot[SlotIndex].Middle = RED THEN
			Station.ColorCount[0] := Station.ColorCount[0] + 1;
		END_IF
		IF Sorter.Slot[SlotIndex].Right = RED THEN
			Station.ColorCount[0] := Station.ColorCount[0] + 1;
		END_IF
		IF Sorter.Slot[SlotIndex].Left = BLACK THEN
			Station.ColorCount[1] := Station.ColorCount[1] + 1;
		END_IF
		IF Sorter.Slot[SlotIndex].Middle = BLACK THEN
			Station.ColorCount[1] := Station.ColorCount[1] + 1;
		END_IF
		IF Sorter.Slot[SlotIndex].Right = BLACK THEN
			Station.ColorCount[1] := Station.ColorCount[1] + 1;
		END_IF
		IF Sorter.Slot[SlotIndex].Left = METALLIC THEN
			Station.ColorCount[2] := Station.ColorCount[2] + 1;
		END_IF
		IF Sorter.Slot[SlotIndex].Middle = METALLIC THEN
			Station.ColorCount[2] := Station.ColorCount[2] + 1;
		END_IF
		IF Sorter.Slot[SlotIndex].Right = METALLIC THEN
			Station.ColorCount[2] := Station.ColorCount[2] + 1;
		END_IF
	END_FOR;

END_ACTION
```

#### OpcUa.st
```iecst
(*********************************************************************************
 * Copyright: I-Automation
 * Author:    John Lee
 * Created:   March 15, 2019/1:21 AM
 *            Opcua setter, reads commands periodically and writes when
*             local state has been changed
 *********************************************************************************)

ACTION OpcUa:

	//Opcua state check timer.
	TON_10ms_Opc.IN := TRUE;
	TON_10ms_Opc.PT := 50;

	//Checks if state has been changed.
	FOR MIndex := 0 TO 7 BY 1 DO
		IF MachineState[MIndex] <> MachineStateOld[MIndex] THEN
			MchUpdate := TRUE;
		END_IF
	END_FOR;

	//If read command finished, update local state
	IF EDGENEG(Station.OpcUa.Read) THEN
		IF MchUpdate = FALSE THEN
			MachineState := OpcUaComm;
		END_IF
	END_IF

	//Opcua Updater
	IF TON_10ms_Opc.Q THEN
		IF MchUpdate THEN
			Station.OpcUa.Write := TRUE;
			MchUpdate := FALSE;
		ELSE
			Station.OpcUa.Read := TRUE;
		END_IF
		TON_10ms_Opc.IN := FALSE;
	END_IF

	//Func block calls
	MachineStateOld := MachineState;
	TON_10ms_Opc();

END_ACTION
```

### Program Logical/Sorting/Machine/SortingStation (IEC) - Sorting conveyor

#### Cyclic.ld - Cyclic code
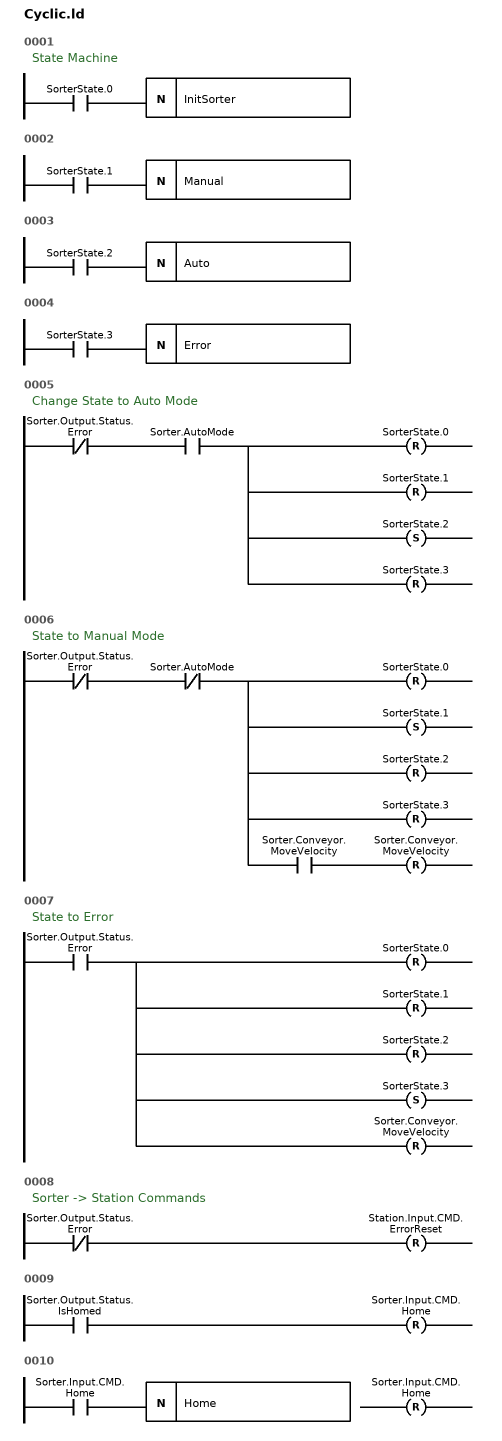
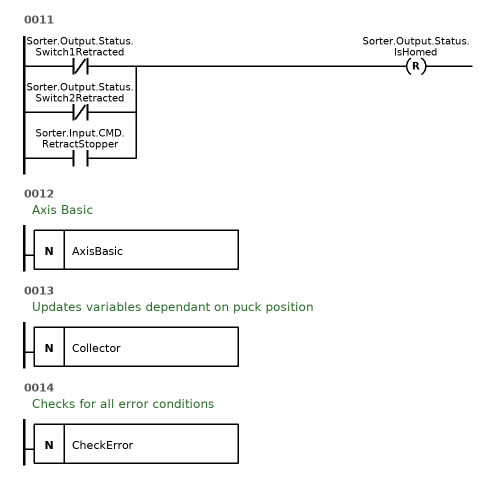
Ladder, written as Structured Text:
```iecst
(*********************************************************************************
 * Copyright: 	I-Automation
 * Author:    	John Lee
 * Created:   	March 8, 2019/12:43 PM
 * Description:    	Private Sorter Control Task
 *********************************************************************************)
 PROGRAM _CYCLIC
VAR
    _p1 : BOOL;
    _p2 : BOOL;
END_VAR
(* Network 1: State Machine  *)
IF SorterState.0 THEN InitSorter; END_IF;

(* Network 2 *)
IF SorterState.1 THEN Manual; END_IF;

(* Network 3 *)
IF SorterState.2 THEN Auto; END_IF;

(* Network 4 *)
IF SorterState.3 THEN Error; END_IF;

(* Network 5: Change State to Auto Mode *)
_p1 := NOT Sorter.Output.Status.Error AND Sorter.AutoMode;
IF _p1 THEN
    SorterState.0 := FALSE;
    SorterState.1 := FALSE;
    SorterState.2 := TRUE;
    SorterState.3 := FALSE;
END_IF;

(* Network 6: State to Manual Mode *)
_p2 := NOT Sorter.Output.Status.Error AND NOT Sorter.AutoMode;
IF _p2 THEN
    SorterState.0 := FALSE;
    SorterState.1 := TRUE;
    SorterState.2 := FALSE;
    SorterState.3 := FALSE;
END_IF;
IF _p2 AND Sorter.Conveyor.MoveVelocity THEN Sorter.Conveyor.MoveVelocity := FALSE; END_IF;

(* Network 7: State to Error  *)
IF Sorter.Output.Status.Error THEN
    SorterState.0 := FALSE;
    SorterState.1 := FALSE;
    SorterState.2 := FALSE;
    SorterState.3 := TRUE;
    Sorter.Conveyor.MoveVelocity := FALSE;
END_IF;

(* Network 8: Sorter -> Station Commands *)
IF NOT Sorter.Output.Status.Error THEN Station.Input.CMD.ErrorReset := FALSE; END_IF;

(* Network 9 *)
IF Sorter.Output.Status.IsHomed THEN Sorter.Input.CMD.Home := FALSE; END_IF;

(* Network 10 *)
IF Sorter.Input.CMD.Home THEN Home; END_IF;
(* never executed: Sorter.Input.CMD.Home := FALSE; *)

(* Network 11 *)
IF NOT Sorter.Output.Status.Switch1Retracted OR NOT Sorter.Output.Status.Switch2Retracted OR Sorter.Input.CMD.RetractStopper THEN
    Sorter.Output.Status.IsHomed := FALSE;
END_IF;

(* Network 12: Axis Basic  *)
AxisBasic;

(* Network 13: Updates variables dependant on puck position *)
Collector;

(* Network 14: Checks for all error conditions *)
CheckError;
END_PROGRAM
```

#### Init.ld - Initialization code
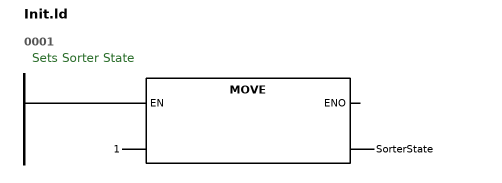
Ladder, written as Structured Text:
```iecst
PROGRAM _INIT
(* Network 1: Sets Sorter State *)
SorterState := 1;
END_PROGRAM
```

#### State.var - Local variables
```iecst
VAR
	AutoState : USINT := 1; (*Automatic state*)
	SorterState : USINT; (*Sorter state*)
	EqLeft : BOOL; (*Equal to left*)
	EqRight : BOOL; (*Equal to right*)
	EqMiddle : BOOL; (*Equal to middle*)
	TON_10ms_Switch1 : TON_10ms; (*Timer value for switch 1*)
	TON_10ms_Switch2 : TON_10ms; (*Timer value for switch 2*)
	TON_10ms_AutoTicker : TON_10ms; (*Auto-ticker timer*)
	TON_10ms_Convey : TON_10ms; (*Timer for convey*)
END_VAR
```

#### Package Logical/Sorting/Machine/SortingStation/States - States

#### InitSorter.ld
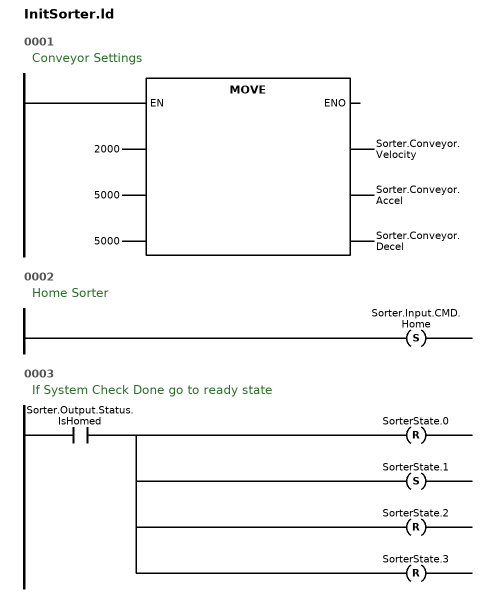
Ladder, written as Structured Text:
```iecst
ACTION InitSorter:
(* Network 1: Conveyor Settings *)
Sorter.Conveyor.Velocity := 2000;
Sorter.Conveyor.Accel := 5000;
Sorter.Conveyor.Decel := 5000;

(* Network 2: Home Sorter *)
Sorter.Input.CMD.Home := TRUE;

(* Network 3: If System Check Done go to ready state *)
IF Sorter.Output.Status.IsHomed THEN
    SorterState.0 := FALSE;
    SorterState.1 := TRUE;
    SorterState.2 := FALSE;
    SorterState.3 := FALSE;
END_IF;
END_ACTION
```

#### Manual.ld
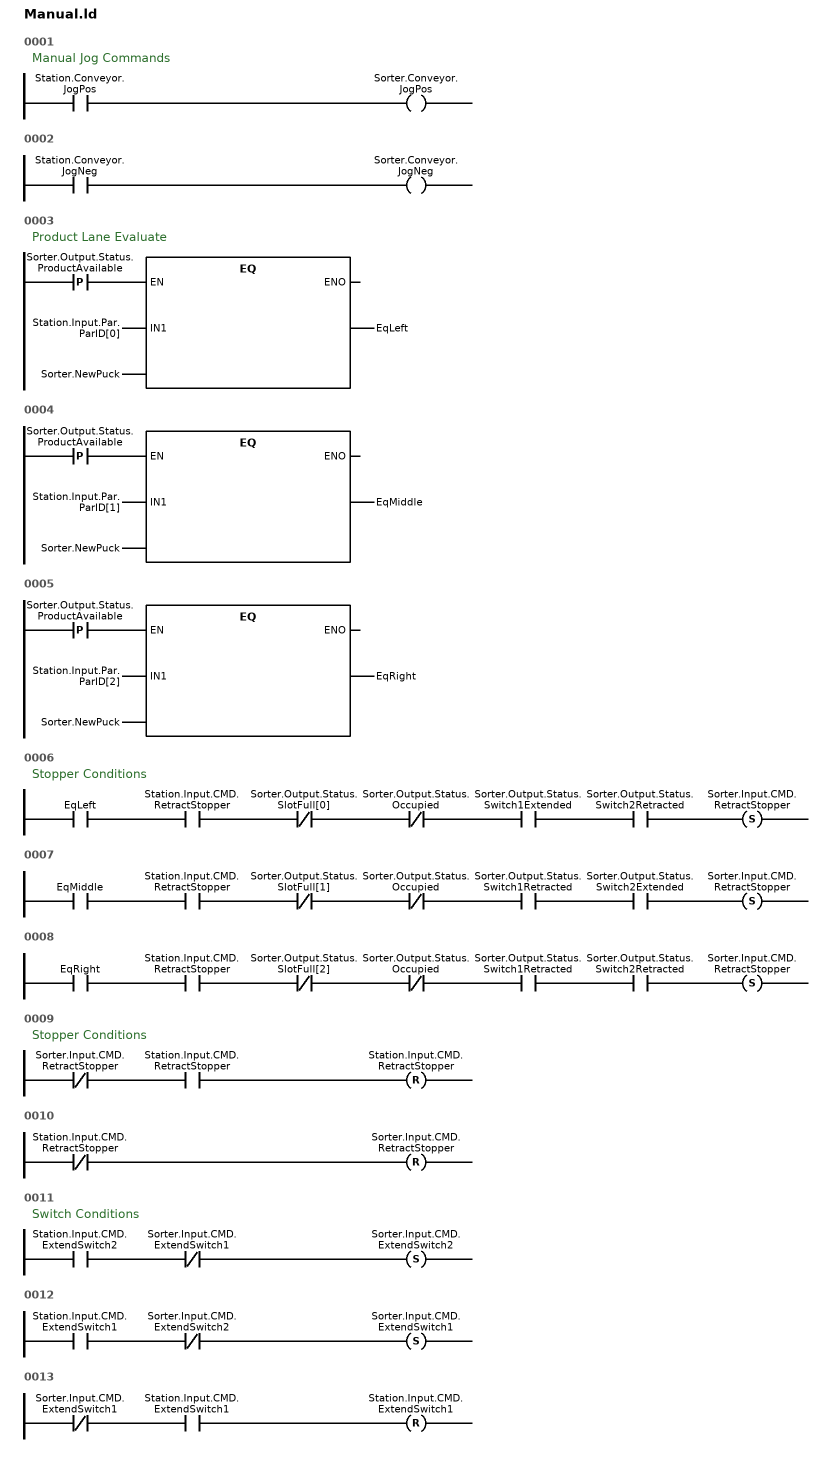
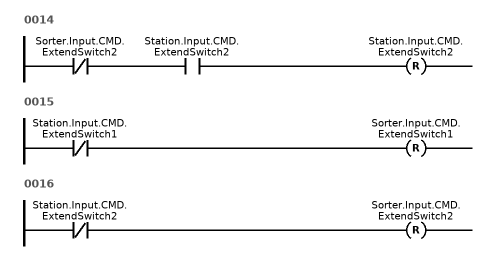
Ladder, written as Structured Text:
```iecst
ACTION Manual:
VAR
    _e1 : R_TRIG;
    _e2 : R_TRIG;
    _e3 : R_TRIG;
END_VAR
(* Network 1: Manual Jog Commands *)
Sorter.Conveyor.JogPos := Station.Conveyor.JogPos;

(* Network 2 *)
Sorter.Conveyor.JogNeg := Station.Conveyor.JogNeg;

(* Network 3: Product Lane Evaluate *)
_e1(CLK := Sorter.Output.Status.ProductAvailable);
IF _e1.Q THEN EqLeft := Station.Input.Par.ParID[0] = Sorter.NewPuck; END_IF;

(* Network 4 *)
_e2(CLK := Sorter.Output.Status.ProductAvailable);
IF _e2.Q THEN EqMiddle := Station.Input.Par.ParID[1] = Sorter.NewPuck; END_IF;

(* Network 5 *)
_e3(CLK := Sorter.Output.Status.ProductAvailable);
IF _e3.Q THEN EqRight := Station.Input.Par.ParID[2] = Sorter.NewPuck; END_IF;

(* Network 6: Stopper Conditions *)
IF EqLeft AND Station.Input.CMD.RetractStopper AND NOT Sorter.Output.Status.SlotFull[0] AND NOT Sorter.Output.Status.Occupied AND Sorter.Output.Status.Switch1Extended AND Sorter.Output.Status.Switch2Retracted THEN
    Sorter.Input.CMD.RetractStopper := TRUE;
END_IF;

(* Network 7 *)
IF EqMiddle AND Station.Input.CMD.RetractStopper AND NOT Sorter.Output.Status.SlotFull[1] AND NOT Sorter.Output.Status.Occupied AND Sorter.Output.Status.Switch1Retracted AND Sorter.Output.Status.Switch2Extended THEN
    Sorter.Input.CMD.RetractStopper := TRUE;
END_IF;

(* Network 8 *)
IF EqRight AND Station.Input.CMD.RetractStopper AND NOT Sorter.Output.Status.SlotFull[2] AND NOT Sorter.Output.Status.Occupied AND Sorter.Output.Status.Switch1Retracted AND Sorter.Output.Status.Switch2Retracted THEN
    Sorter.Input.CMD.RetractStopper := TRUE;
END_IF;

(* Network 9: Stopper Conditions *)
IF NOT Sorter.Input.CMD.RetractStopper AND Station.Input.CMD.RetractStopper THEN
    Station.Input.CMD.RetractStopper := FALSE;
END_IF;

(* Network 10 *)
IF NOT Station.Input.CMD.RetractStopper THEN Sorter.Input.CMD.RetractStopper := FALSE; END_IF;

(* Network 11: Switch Conditions *)
IF Station.Input.CMD.ExtendSwitch2 AND NOT Sorter.Input.CMD.ExtendSwitch1 THEN
    Sorter.Input.CMD.ExtendSwitch2 := TRUE;
END_IF;

(* Network 12 *)
IF Station.Input.CMD.ExtendSwitch1 AND NOT Sorter.Input.CMD.ExtendSwitch2 THEN
    Sorter.Input.CMD.ExtendSwitch1 := TRUE;
END_IF;

(* Network 13 *)
IF NOT Sorter.Input.CMD.ExtendSwitch1 AND Station.Input.CMD.ExtendSwitch1 THEN
    Station.Input.CMD.ExtendSwitch1 := FALSE;
END_IF;

(* Network 14 *)
IF NOT Sorter.Input.CMD.ExtendSwitch2 AND Station.Input.CMD.ExtendSwitch2 THEN
    Station.Input.CMD.ExtendSwitch2 := FALSE;
END_IF;

(* Network 15 *)
IF NOT Station.Input.CMD.ExtendSwitch1 THEN Sorter.Input.CMD.ExtendSwitch1 := FALSE; END_IF;

(* Network 16 *)
IF NOT Station.Input.CMD.ExtendSwitch2 THEN Sorter.Input.CMD.ExtendSwitch2 := FALSE; END_IF;
END_ACTION
```

#### Auto.ld
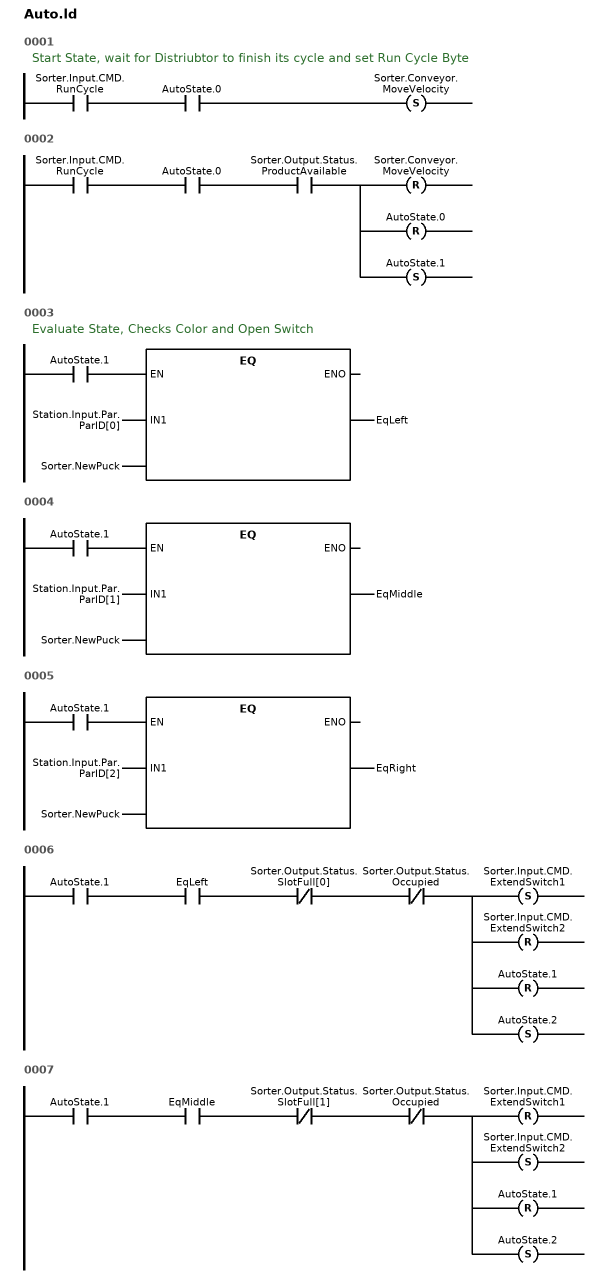
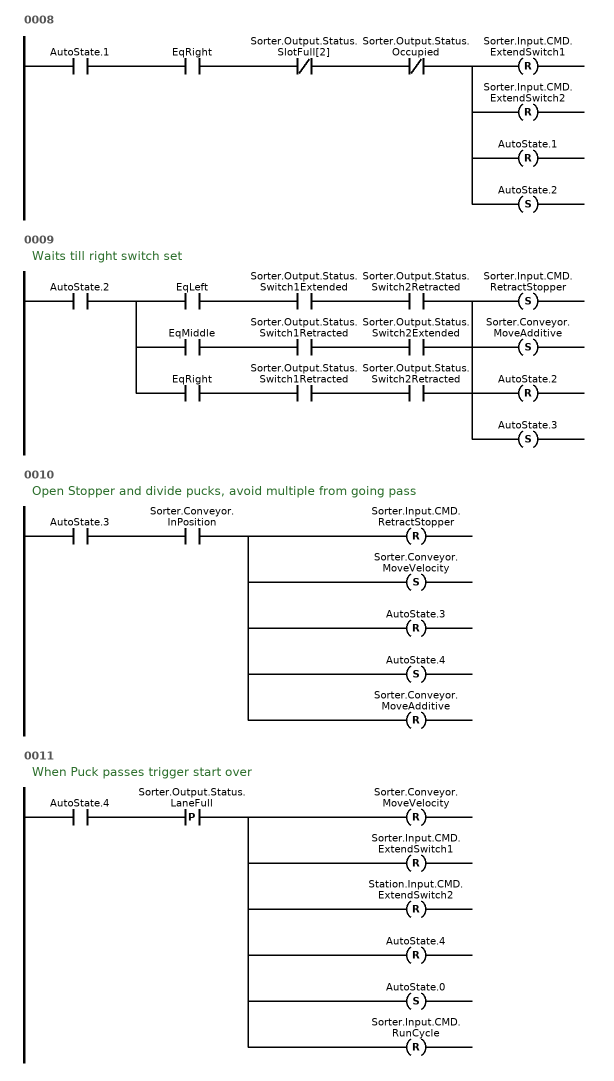
Ladder, written as Structured Text:
```iecst
ACTION Auto:
VAR
    _p1 : BOOL;
    _p2 : BOOL;
    _p3 : BOOL;
    _p4 : BOOL;
    _p5 : BOOL;
    _p6 : BOOL;
    _p7 : BOOL;
    _p8 : BOOL;
    _e9 : R_TRIG;
    _p10 : BOOL;
END_VAR
(* Network 1: Start State, wait for Distriubtor to finish its cycle and set Run Cycle Byte *)
IF Sorter.Input.CMD.RunCycle AND AutoState.0 THEN Sorter.Conveyor.MoveVelocity := TRUE; END_IF;

(* Network 2 *)
_p1 := Sorter.Input.CMD.RunCycle AND AutoState.0 AND Sorter.Output.Status.ProductAvailable;
IF _p1 THEN
    Sorter.Conveyor.MoveVelocity := FALSE;
    AutoState.0 := FALSE;
    AutoState.1 := TRUE;
END_IF;

(* Network 3: Evaluate State, Checks Color and Open Switch *)
IF AutoState.1 THEN EqLeft := Station.Input.Par.ParID[0] = Sorter.NewPuck; END_IF;

(* Network 4 *)
IF AutoState.1 THEN EqMiddle := Station.Input.Par.ParID[1] = Sorter.NewPuck; END_IF;

(* Network 5 *)
IF AutoState.1 THEN EqRight := Station.Input.Par.ParID[2] = Sorter.NewPuck; END_IF;

(* Network 6 *)
_p2 := AutoState.1 AND EqLeft AND NOT Sorter.Output.Status.SlotFull[0] AND NOT Sorter.Output.Status.Occupied;
IF _p2 THEN
    Sorter.Input.CMD.ExtendSwitch1 := TRUE;
    Sorter.Input.CMD.ExtendSwitch2 := FALSE;
    AutoState.1 := FALSE;
    AutoState.2 := TRUE;
END_IF;

(* Network 7 *)
_p3 := AutoState.1 AND EqMiddle AND NOT Sorter.Output.Status.SlotFull[1] AND NOT Sorter.Output.Status.Occupied;
IF _p3 THEN
    Sorter.Input.CMD.ExtendSwitch1 := FALSE;
    Sorter.Input.CMD.ExtendSwitch2 := TRUE;
    AutoState.1 := FALSE;
    AutoState.2 := TRUE;
END_IF;

(* Network 8 *)
_p4 := AutoState.1 AND EqRight AND NOT Sorter.Output.Status.SlotFull[2] AND NOT Sorter.Output.Status.Occupied;
IF _p4 THEN
    Sorter.Input.CMD.ExtendSwitch1 := FALSE;
    Sorter.Input.CMD.ExtendSwitch2 := FALSE;
    AutoState.1 := FALSE;
    AutoState.2 := TRUE;
END_IF;

(* Network 9: Waits till right switch set *)
_p5 := AutoState.2 AND EqLeft AND Sorter.Output.Status.Switch1Extended AND Sorter.Output.Status.Switch2Retracted;
_p6 := AutoState.2 AND EqMiddle AND Sorter.Output.Status.Switch1Retracted AND Sorter.Output.Status.Switch2Extended;
_p7 := AutoState.2 AND EqRight AND Sorter.Output.Status.Switch1Retracted AND Sorter.Output.Status.Switch2Retracted;
IF _p5 OR _p6 OR _p7 THEN
    Sorter.Input.CMD.RetractStopper := TRUE;
    Sorter.Conveyor.MoveAdditive := TRUE;
    AutoState.2 := FALSE;
    AutoState.3 := TRUE;
END_IF;

(* Network 10: Open Stopper and divide pucks, avoid multiple from going pass *)
_p8 := AutoState.3 AND Sorter.Conveyor.InPosition;
IF AutoState.3 AND Sorter.Conveyor.InPosition THEN Sorter.Input.CMD.RetractStopper := FALSE; END_IF;
IF _p8 THEN
    Sorter.Conveyor.MoveVelocity := TRUE;
    AutoState.3 := FALSE;
    AutoState.4 := TRUE;
    Sorter.Conveyor.MoveAdditive := FALSE;
END_IF;

(* Network 11: When Puck passes trigger start over *)
_e9(CLK := Sorter.Output.Status.LaneFull);
IF AutoState.4 AND _e9.Q THEN
    Sorter.Conveyor.MoveVelocity := FALSE;
    Sorter.Input.CMD.ExtendSwitch1 := FALSE;
    Station.Input.CMD.ExtendSwitch2 := FALSE;
END_IF;
_p10 := AutoState.4 AND _e9.Q;
IF AutoState.4 AND _e9.Q THEN AutoState.4 := FALSE; END_IF;
IF _p10 THEN
    AutoState.0 := TRUE;
    Sorter.Input.CMD.RunCycle := FALSE;
END_IF;
END_ACTION
```

#### Error.ld
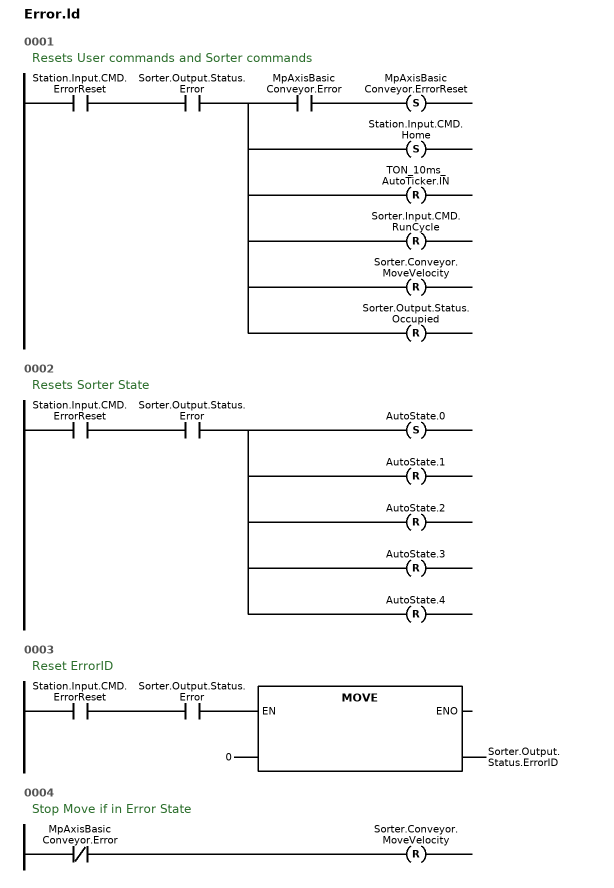
Ladder, written as Structured Text:
```iecst
ACTION Error:
VAR
    _p1 : BOOL;
    _p2 : BOOL;
    _p3 : BOOL;
END_VAR
(* Network 1: Resets User commands and Sorter commands *)
_p1 := Station.Input.CMD.ErrorReset AND Sorter.Output.Status.Error;
IF _p1 AND MpAxisBasicConveyor.Error THEN MpAxisBasicConveyor.ErrorReset := TRUE; END_IF;
IF _p1 THEN
    Station.Input.CMD.Home := TRUE;
    TON_10ms_AutoTicker.IN := FALSE;
    Sorter.Input.CMD.RunCycle := FALSE;
    Sorter.Conveyor.MoveVelocity := FALSE;
    Sorter.Output.Status.Occupied := FALSE;
END_IF;

(* Network 2: Resets Sorter State *)
_p2 := Station.Input.CMD.ErrorReset AND Sorter.Output.Status.Error;
IF _p2 THEN
    AutoState.0 := TRUE;
    AutoState.1 := FALSE;
    AutoState.2 := FALSE;
    AutoState.3 := FALSE;
    AutoState.4 := FALSE;
END_IF;

(* Network 3: Reset ErrorID *)
_p3 := Station.Input.CMD.ErrorReset AND Sorter.Output.Status.Error;
IF _p3 THEN Sorter.Output.Status.ErrorID := 0; END_IF;

(* Network 4: Stop Move if in Error State *)
IF NOT MpAxisBasicConveyor.Error THEN Sorter.Conveyor.MoveVelocity := FALSE; END_IF;
END_ACTION
```

#### Package Logical/Sorting/Machine/SortingStation/Actions - Actions

#### Home.ld
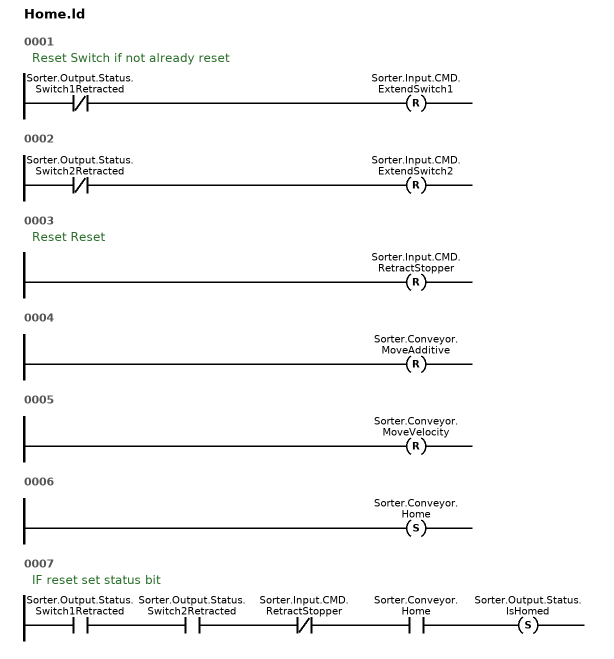
Ladder, written as Structured Text:
```iecst
ACTION Home:
(* Network 1: Reset Switch if not already reset *)
IF NOT Sorter.Output.Status.Switch1Retracted THEN Sorter.Input.CMD.ExtendSwitch1 := FALSE; END_IF;

(* Network 2 *)
IF NOT Sorter.Output.Status.Switch2Retracted THEN Sorter.Input.CMD.ExtendSwitch2 := FALSE; END_IF;

(* Network 3: Reset Reset *)
Sorter.Input.CMD.RetractStopper := FALSE;

(* Network 4 *)
Sorter.Conveyor.MoveAdditive := FALSE;

(* Network 5 *)
Sorter.Conveyor.MoveVelocity := FALSE;

(* Network 6 *)
Sorter.Conveyor.Home := TRUE;

(* Network 7: IF reset set status bit *)
IF Sorter.Output.Status.Switch1Retracted AND Sorter.Output.Status.Switch2Retracted AND NOT Sorter.Input.CMD.RetractStopper AND Sorter.Conveyor.Home THEN
    Sorter.Output.Status.IsHomed := TRUE;
END_IF;
END_ACTION
```

#### AxisBasic.ld
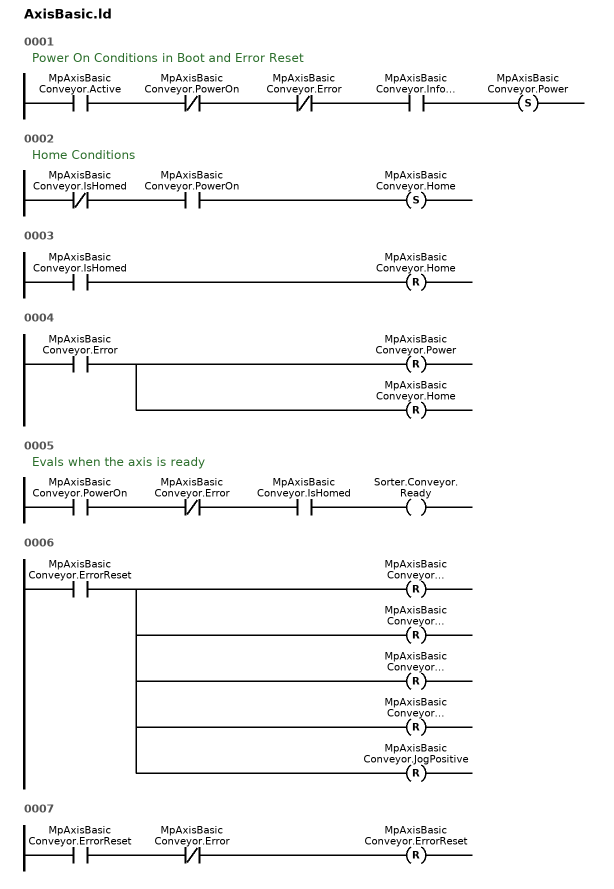
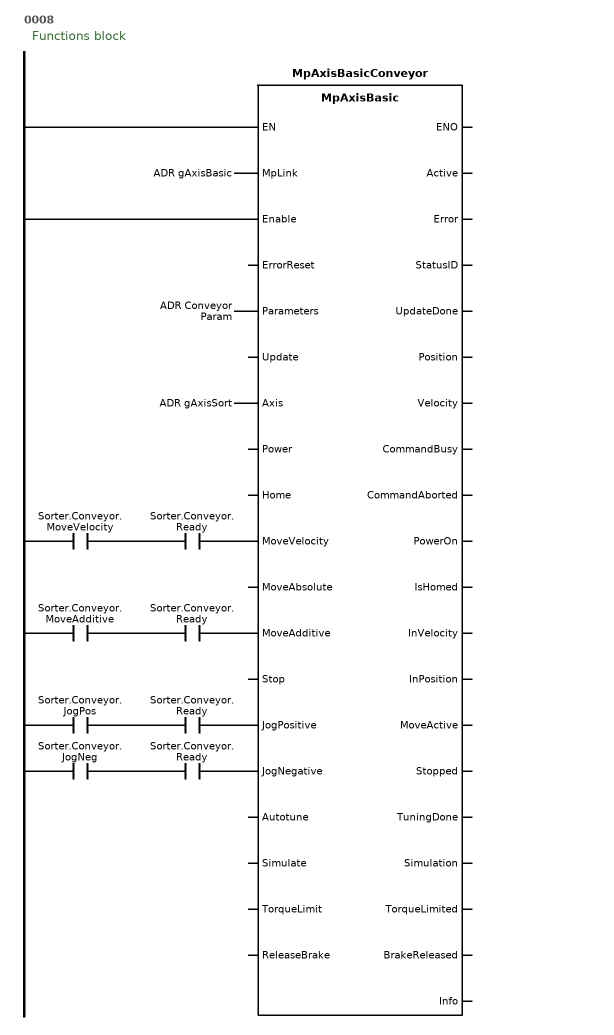
Ladder, written as Structured Text:
```iecst
ACTION AxisBasic:
VAR
    _p1 : BOOL;
    _p2 : BOOL;
END_VAR
(* Network 1: Power On Conditions in Boot and Error Reset *)
IF MpAxisBasicConveyor.Active AND NOT MpAxisBasicConveyor.PowerOn AND NOT MpAxisBasicConveyor.Error AND MpAxisBasicConveyor.Info.ReadyToPowerOn THEN
    MpAxisBasicConveyor.Power := TRUE;
END_IF;

(* Network 2: Home Conditions *)
IF NOT MpAxisBasicConveyor.IsHomed AND MpAxisBasicConveyor.PowerOn THEN
    MpAxisBasicConveyor.Home := TRUE;
END_IF;

(* Network 3 *)
IF MpAxisBasicConveyor.IsHomed THEN MpAxisBasicConveyor.Home := FALSE; END_IF;

(* Network 4 *)
_p1 := MpAxisBasicConveyor.Error;
IF MpAxisBasicConveyor.Error THEN MpAxisBasicConveyor.Power := FALSE; END_IF;
IF _p1 THEN MpAxisBasicConveyor.Home := FALSE; END_IF;

(* Network 5: Evals when the axis is ready *)
Sorter.Conveyor.Ready := MpAxisBasicConveyor.PowerOn AND NOT MpAxisBasicConveyor.Error AND MpAxisBasicConveyor.IsHomed;

(* Network 6 *)
_p2 := MpAxisBasicConveyor.ErrorReset;
IF MpAxisBasicConveyor.ErrorReset THEN MpAxisBasicConveyor.MoveAdditive := FALSE; END_IF;
IF _p2 THEN
    MpAxisBasicConveyor.MoveVelocity := FALSE;
    MpAxisBasicConveyor.MoveAdditive := FALSE;
    MpAxisBasicConveyor.JogNegative := FALSE;
    MpAxisBasicConveyor.JogPositive := FALSE;
END_IF;

(* Network 7 *)
IF MpAxisBasicConveyor.ErrorReset AND NOT MpAxisBasicConveyor.Error THEN
    MpAxisBasicConveyor.ErrorReset := FALSE;
END_IF;

(* Network 8: Functions block *)
MpAxisBasicConveyor(MpLink := ADR(gAxisBasic), Enable := TRUE, Parameters := ADR(ConveyorParam), Axis := ADR(gAxisSort), MoveVelocity := Sorter.Conveyor.MoveVelocity AND Sorter.Conveyor.Ready, MoveAdditive := Sorter.Conveyor.MoveAdditive AND Sorter.Conveyor.Ready, JogPositive := Sorter.Conveyor.JogPos AND Sorter.Conveyor.Ready, JogNegative := Sorter.Conveyor.JogNeg AND Sorter.Conveyor.Ready);
END_ACTION
```

#### Collector.ld
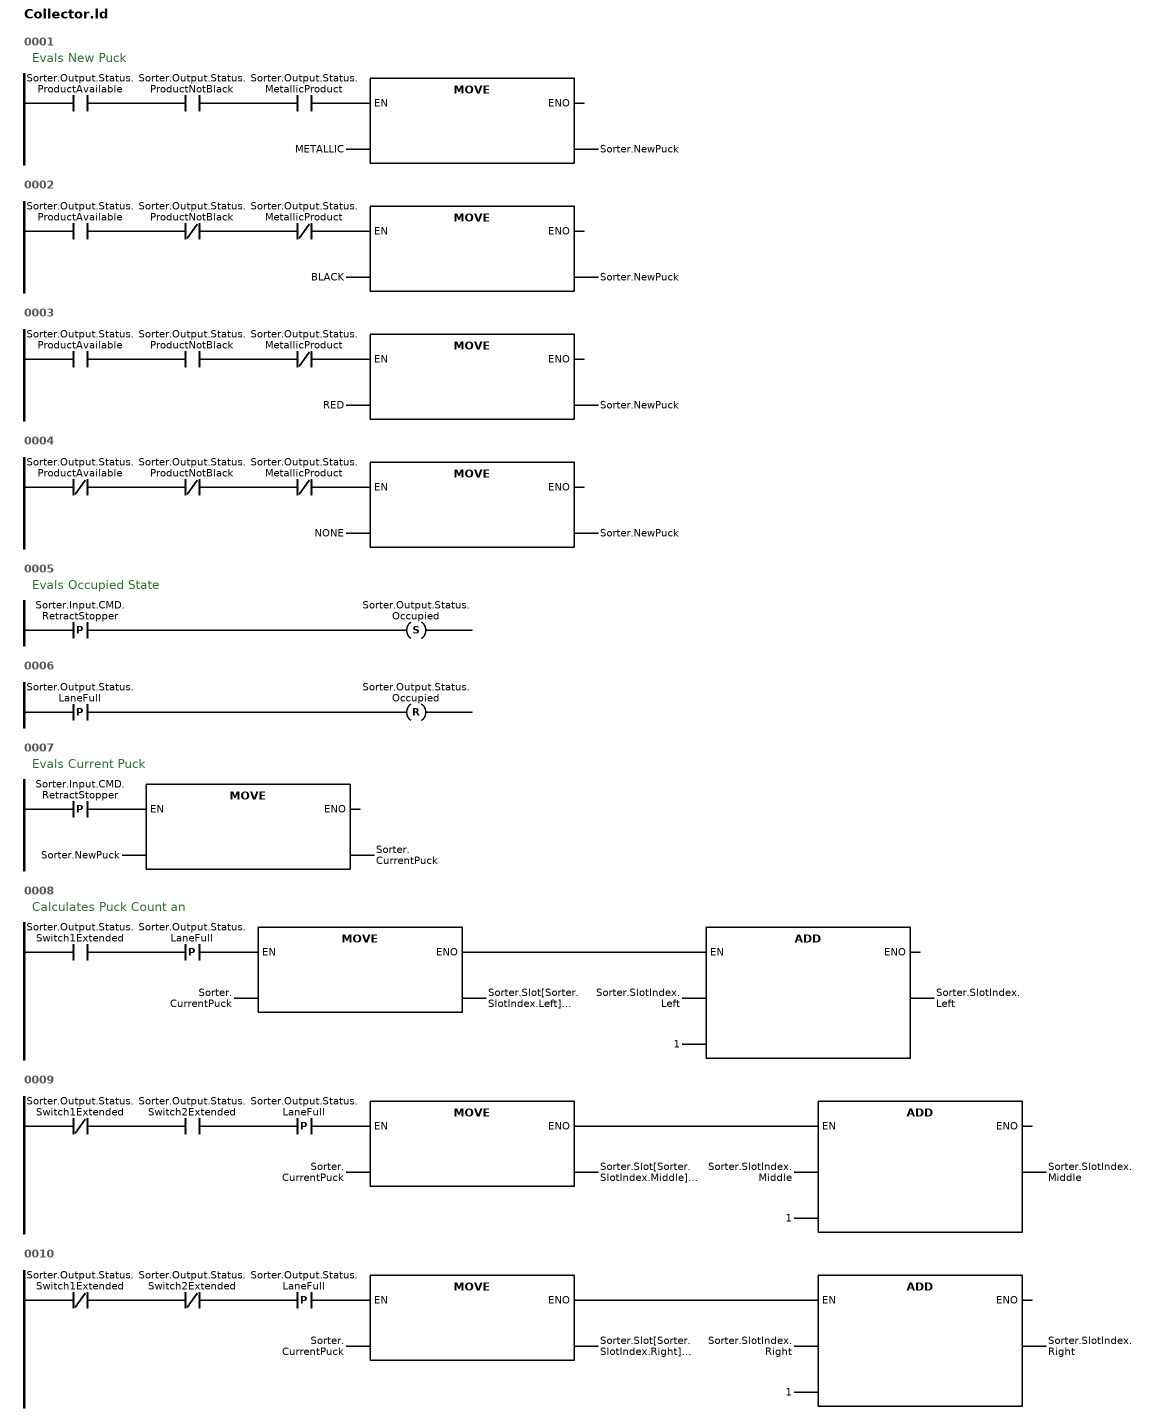
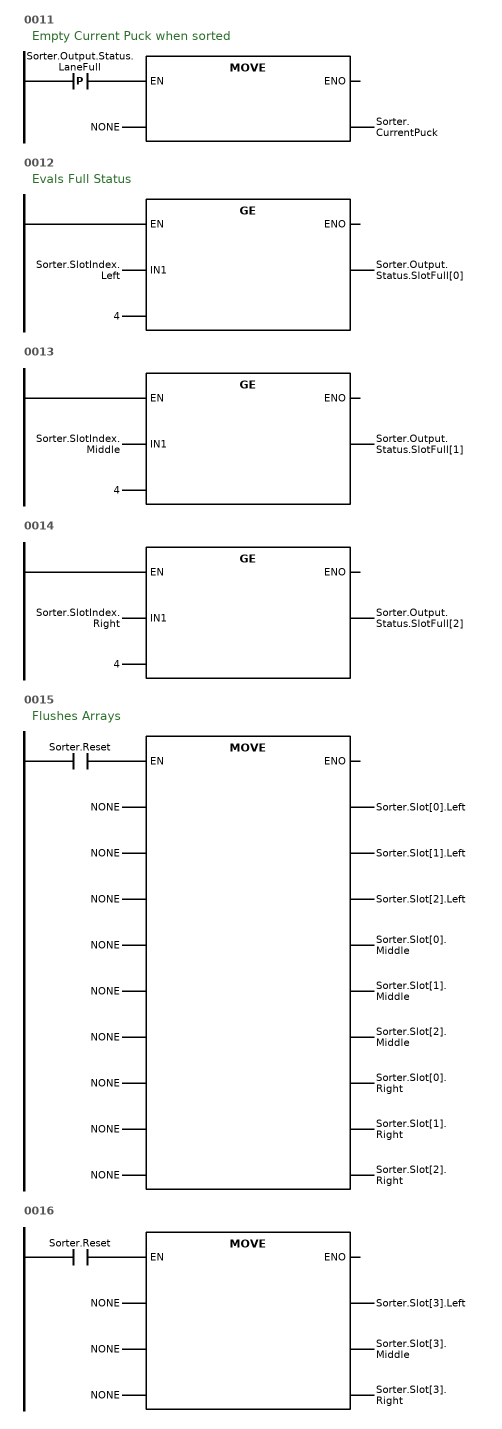
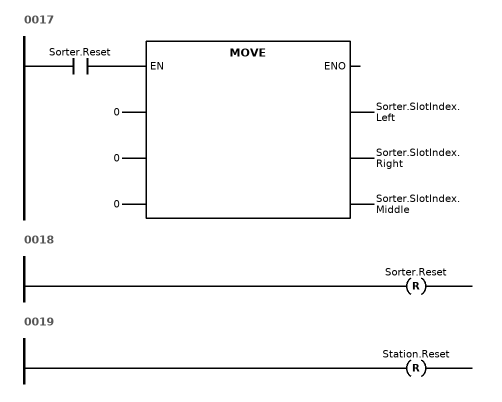
Ladder, written as Structured Text:
```iecst
ACTION Collector:
VAR
    _p1 : BOOL;
    _p2 : BOOL;
    _p3 : BOOL;
    _p4 : BOOL;
    _e5 : R_TRIG;
    _e6 : R_TRIG;
    _e7 : R_TRIG;
    _e8 : R_TRIG;
    _p9 : BOOL;
    _e10 : R_TRIG;
    _p11 : BOOL;
    _e12 : R_TRIG;
    _p13 : BOOL;
    _e14 : R_TRIG;
    _p15 : BOOL;
    _p16 : BOOL;
    _p17 : BOOL;
END_VAR
(* Network 1: Evals New Puck *)
_p1 := Sorter.Output.Status.ProductAvailable AND Sorter.Output.Status.ProductNotBlack AND Sorter.Output.Status.MetallicProduct;
IF _p1 THEN Sorter.NewPuck := METALLIC; END_IF;

(* Network 2 *)
_p2 := Sorter.Output.Status.ProductAvailable AND NOT Sorter.Output.Status.ProductNotBlack AND NOT Sorter.Output.Status.MetallicProduct;
IF _p2 THEN Sorter.NewPuck := BLACK; END_IF;

(* Network 3 *)
_p3 := Sorter.Output.Status.ProductAvailable AND Sorter.Output.Status.ProductNotBlack AND NOT Sorter.Output.Status.MetallicProduct;
IF _p3 THEN Sorter.NewPuck := RED; END_IF;

(* Network 4 *)
_p4 := NOT Sorter.Output.Status.ProductAvailable AND NOT Sorter.Output.Status.ProductNotBlack AND NOT Sorter.Output.Status.MetallicProduct;
IF _p4 THEN Sorter.NewPuck := NONE; END_IF;

(* Network 5: Evals Occupied State *)
_e5(CLK := Sorter.Input.CMD.RetractStopper);
IF _e5.Q THEN Sorter.Output.Status.Occupied := TRUE; END_IF;

(* Network 6 *)
_e6(CLK := Sorter.Output.Status.LaneFull);
IF _e6.Q THEN Sorter.Output.Status.Occupied := FALSE; END_IF;

(* Network 7: Evals Current Puck *)
_e7(CLK := Sorter.Input.CMD.RetractStopper);
IF _e7.Q THEN Sorter.CurrentPuck := Sorter.NewPuck; END_IF;

(* Network 8: Calculates Puck Count an *)
_e8(CLK := Sorter.Output.Status.LaneFull);
_p9 := Sorter.Output.Status.Switch1Extended AND _e8.Q;
IF _p9 THEN
    Sorter.Slot[Sorter.SlotIndex.Left].Left := Sorter.CurrentPuck;
    Sorter.SlotIndex.Left := Sorter.SlotIndex.Left + 1;
END_IF;

(* Network 9 *)
_e10(CLK := Sorter.Output.Status.LaneFull);
_p11 := NOT Sorter.Output.Status.Switch1Extended AND Sorter.Output.Status.Switch2Extended AND _e10.Q;
IF _p11 THEN
    Sorter.Slot[Sorter.SlotIndex.Middle].Middle := Sorter.CurrentPuck;
    Sorter.SlotIndex.Middle := Sorter.SlotIndex.Middle + 1;
END_IF;

(* Network 10 *)
_e12(CLK := Sorter.Output.Status.LaneFull);
_p13 := NOT Sorter.Output.Status.Switch1Extended AND NOT Sorter.Output.Status.Switch2Extended AND _e12.Q;
IF _p13 THEN
    Sorter.Slot[Sorter.SlotIndex.Right].Right := Sorter.CurrentPuck;
    Sorter.SlotIndex.Right := Sorter.SlotIndex.Right + 1;
END_IF;

(* Network 11: Empty Current Puck when sorted *)
_e14(CLK := Sorter.Output.Status.LaneFull);
IF _e14.Q THEN Sorter.CurrentPuck := NONE; END_IF;

(* Network 12: Evals Full Status *)
Sorter.Output.Status.SlotFull[0] := Sorter.SlotIndex.Left >= 4;

(* Network 13 *)
Sorter.Output.Status.SlotFull[1] := Sorter.SlotIndex.Middle >= 4;

(* Network 14 *)
Sorter.Output.Status.SlotFull[2] := Sorter.SlotIndex.Right >= 4;

(* Network 15: Flushes Arrays *)
_p15 := Sorter.Reset;
IF _p15 THEN
    Sorter.Slot[0].Left := NONE;
    Sorter.Slot[1].Left := NONE;
    Sorter.Slot[2].Left := NONE;
    Sorter.Slot[0].Middle := NONE;
    Sorter.Slot[1].Middle := NONE;
    Sorter.Slot[2].Middle := NONE;
    Sorter.Slot[0].Right := NONE;
    Sorter.Slot[1].Right := NONE;
    Sorter.Slot[2].Right := NONE;
END_IF;

(* Network 16 *)
_p16 := Sorter.Reset;
IF _p16 THEN
    Sorter.Slot[3].Left := NONE;
    Sorter.Slot[3].Middle := NONE;
    Sorter.Slot[3].Right := NONE;
END_IF;

(* Network 17 *)
_p17 := Sorter.Reset;
IF _p17 THEN
    Sorter.SlotIndex.Left := 0;
    Sorter.SlotIndex.Right := 0;
    Sorter.SlotIndex.Middle := 0;
END_IF;

(* Network 18 *)
Sorter.Reset := FALSE;

(* Network 19 *)
Station.Reset := FALSE;
END_ACTION
```

#### CheckError.st
```iecst
(*********************************************************************************
 * Copyright: I-Automation
 * Author:    John Lee
 * Created:   March 15, 2019/1:48 AM
 *  		  Error Checking Task for
 *-------------------------------------------
   Rejection Codes:
 * 0 Nothing Wrong
 * 10 Switch2 Not Retracted
 * 20 Switch1 Not Retracted
 * 30 Left Lane Full
 * 31 Switch 1 Retracted
 * 32 Middle Lane Full
 * 33 Switch 2 Retracted
 * 34 Right Lane Full
 * 36 Station is Occupied
 * 37 No Puck Detected
 * 38 Switch 1 Extended
 * 39 Switch 2 Exnteded
 *--------------------------------------------
  Error Codes:
 * 0 No Error
 * 1 Left Lane Full
 * 2 Middle Lane Full
 * 3 Right Lane Full
 * 4 No Product Availiable
 * 5 Switch is Stuck
 * 6 Puck Missing
 * 7 Axis Error
 *********************************************************************************)

ACTION CheckError:

	TON_10ms_Switch1.PT    :=  400;  //Error timer for Switch 1
	TON_10ms_Switch2.PT    :=  400;  //Error timer for Switch 2
	TON_10ms_AutoTicker.PT :=  1000; //Error timer for transitioning between states

	Sorter.Output.RejectionCode   := 0;		//Resetings Rejection Code
	Sorter.Output.CommandRejected := FALSE;

	CASE SorterState OF

		2:  // Manual Mode Error Check

			// Rejection Conditions for Switch 1
			IF Station.Input.CMD.ExtendSwitch1 THEN
				IF Sorter.Output.Status.Switch1Extended THEN
					TON_10ms_Switch1.IN := FALSE;
				ELSIF Sorter.Output.Status.Switch2Extended THEN
					Sorter.Output.RejectionCode := 10;
					Sorter.Output.CommandRejected := TRUE;
				ELSE
					TON_10ms_Switch1.IN := TRUE;
				END_IF
			END_IF

			//Rejection Conditions for Switch 2
			IF Station.Input.CMD.ExtendSwitch2 THEN
				IF Sorter.Output.Status.Switch2Extended THEN
					TON_10ms_Switch2.IN := FALSE;
				ELSIF Sorter.Output.Status.Switch1Extended THEN
					Sorter.Output.RejectionCode := 20;
					Sorter.Output.CommandRejected := TRUE;
				ELSE
					TON_10ms_Switch2.IN := TRUE;
				END_IF
			END_IF

			//Rejection Conditions for Stopper
			IF Station.Input.CMD.RetractStopper THEN
				//Left Lane
				IF Sorter.NewPuck = Sorter.Input.Par.ParID[0] THEN
					IF Sorter.Output.Status.SlotFull[0] THEN
						Sorter.Output.RejectionCode := 30;    		//Left Slow Full
						Sorter.Output.CommandRejected := TRUE;
					END_IF
					IF Sorter.Output.Status.Switch1Retracted THEN
						Sorter.Output.RejectionCode := 31;    		//Switch 1 Not Extended
						Sorter.Output.CommandRejected := TRUE;
					END_IF
				END_IF
				//Middle Lane
				IF Sorter.NewPuck = Sorter.Input.Par.ParID[1] THEN
					IF Sorter.Output.Status.SlotFull[1] THEN
						Sorter.Output.RejectionCode := 32;    		//Left Slow Full
						Sorter.Output.CommandRejected := TRUE;
					END_IF
					IF Sorter.Output.Status.Switch1Extended THEN
						Sorter.Output.RejectionCode := 38;    		//Switch 1 Not Extended
						Sorter.Output.CommandRejected := TRUE;
					END_IF
					IF Sorter.Output.Status.Switch2Retracted THEN
						Sorter.Output.RejectionCode := 33;    		//Switch 1 Not Extended
						Sorter.Output.CommandRejected := TRUE;
					END_IF
				END_IF
				//Right Lane
				IF Sorter.NewPuck = Sorter.Input.Par.ParID[2] THEN
					IF Sorter.Output.Status.SlotFull[2] THEN
						Sorter.Output.RejectionCode := 34;    		//Left Slow Full
						Sorter.Output.CommandRejected := TRUE;
					END_IF
					IF Sorter.Output.Status.Switch1Extended THEN
						Sorter.Output.RejectionCode := 38;    		//Switch 1 Not Extended
						Sorter.Output.CommandRejected := TRUE;
					END_IF
					IF Sorter.Output.Status.Switch2Extended THEN
						Sorter.Output.RejectionCode := 39;    		//Switch 1 Not Extended
						Sorter.Output.CommandRejected := TRUE;
					END_IF
				END_IF
				// No Puck
				IF Sorter.NewPuck = NONE THEN
					Sorter.Output.RejectionCode := 37;        	 //No Puck
					Sorter.Output.CommandRejected := TRUE;
				END_IF
				// If Occupied
				IF Sorter.Output.Status.Occupied THEN
					Sorter.Output.RejectionCode := 36;    		//Switch2 Not Retracted
					Sorter.Output.CommandRejected := TRUE;
				END_IF
			END_IF

		4:

			//Error Condtions for Auto State

			//Init State
			IF AutoState.0 THEN
				IF EDGEPOS(Sorter.Output.Status.LaneFull) THEN
					TON_10ms_AutoTicker.IN := FALSE;
				END_IF

				IF Sorter.Input.CMD.RunCycle THEN
					TON_10ms_AutoTicker.IN := TRUE;
				END_IF
				IF  Sorter.Output.Status.ProductAvailable THEN
					TON_10ms_AutoTicker.IN := FALSE;
				END_IF
			END_IF

			//Classify State
			IF AutoState.1 THEN
				IF EqLeft THEN
					IF Sorter.Output.Status.SlotFull[0] THEN
						Sorter.Output.Status.ErrorID := 1;    		//Left Lane Full
						TON_10ms_AutoTicker.IN := FALSE;
					END_IF
				END_IF
				IF EqMiddle THEN
					IF Sorter.Output.Status.SlotFull[1] THEN
						Sorter.Output.Status.ErrorID := 2;    		//Middle Lane Full
						TON_10ms_AutoTicker.IN := FALSE;
					END_IF
				END_IF
				IF EqRight THEN
					IF Sorter.Output.Status.SlotFull[2] THEN
						Sorter.Output.Status.ErrorID := 3;    		//Right Lane FULL
						TON_10ms_AutoTicker.IN := FALSE;
					END_IF
				END_IF
				IF Sorter.Output.Status.Switch1Extended OR
					Sorter.Output.Status.Switch2Extended THEN
					TON_10ms_AutoTicker.IN := FALSE;
				END_IF
			END_IF

			//Time Out Errors

			//Switch On
			IF AutoState.2 THEN
				TON_10ms_AutoTicker.IN := TRUE;
			END_IF
			//Puck Travel
			IF AutoState.3 THEN
				TON_10ms_AutoTicker.IN := TRUE;
			END_IF
			// Done
			IF AutoState.4 THEN
				TON_10ms_AutoTicker.IN := TRUE;
			END_IF
	END_CASE;

	//Axis Error
	IF MpAxisBasicConveyor.Error THEN
		Sorter.Output.Status.ErrorID := 7;
	END_IF

	//Hardware Module Error
	IF  NOT gSortModuleOK.BusController 	OR
		NOT gSortModuleOK.BusTransmitter 	OR
		NOT gSortModuleOK.DigitalInput 		OR
		NOT gSortModuleOK.DigitalOutput 	OR
		NOT gSortModuleOK.Interface 		OR
		NOT gSortModuleOK.PotentialDist0011 OR
		NOT gSortModuleOK.PotentialDist0012 OR
		NOT gSortModuleOK.PowerSupply 		OR
		NOT gSortModuleOK.StepperMotor 		THEN
		Sorter.Output.Status.ErrorID := 8;
	END_IF

	//Time out Checker
	IF TON_10ms_AutoTicker.Q THEN
		CASE AutoState OF
			1:
				Sorter.Output.Status.ErrorID := 4;  // Product Not Availiable
			2:
				Sorter.Output.Status.ErrorID := 5;	 // Switch Stuck
			4:
				Sorter.Output.Status.ErrorID := 5;	 // Switch Stuck
			8:
				Sorter.Output.Status.ErrorID := 6;  // 404 Puck
			16:
		 		Sorter.Output.Status.ErrorID := 6;  // 404 Puck
		END_CASE;
	END_IF

	//Setting Error Flag
	IF Sorter.Output.Status.ErrorID <> 0 THEN
		Sorter.Output.Status.Error := TRUE;
	ELSE
		Sorter.Output.Status.Error := FALSE;
	END_IF

	//Time Outs for Switches
	IF TON_10ms_Switch1.Q THEN
		Sorter.Output.CommandRejected := TRUE;
		Sorter.Output.RejectionCode := 11;
	END_IF
	IF TON_10ms_Switch2.Q THEN
		Sorter.Output.CommandRejected := TRUE;
		Sorter.Output.RejectionCode := 21;
	END_IF

	TON_10ms_Switch1();
	TON_10ms_Switch2();
	TON_10ms_AutoTicker();
END_ACTION
```

#### CheckError.ld - not listed in the package file held
Ladder, written as Structured Text:
```iecst
ACTION CheckError:
(* Network 1 *)
END_ACTION
```

#### Station.var - not listed in the package file held
```iecst
VAR
	AutoState : USINT := 1;
	SorterState : USINT;
	EqLeft : BOOL;
	EqRight : BOOL;
	EqMiddle : BOOL;
END_VAR
```

### Program Logical/Sorting/Machine/IOCtrl (IEC) - Sorter inputs and outputs

#### Variables.var
```iecst
VAR CONSTANT
	PUCK_PAST : REAL := 400; (*The product has passed*)
END_VAR
VAR
	Update_Accel : BOOL; (*Update acceleration parameter*)
	Update_Decel : BOOL; (*Update deceleration parameter*)
	Update_Vel : BOOL; (*Update velocity*)
END_VAR
```

#### Cyclic.ld
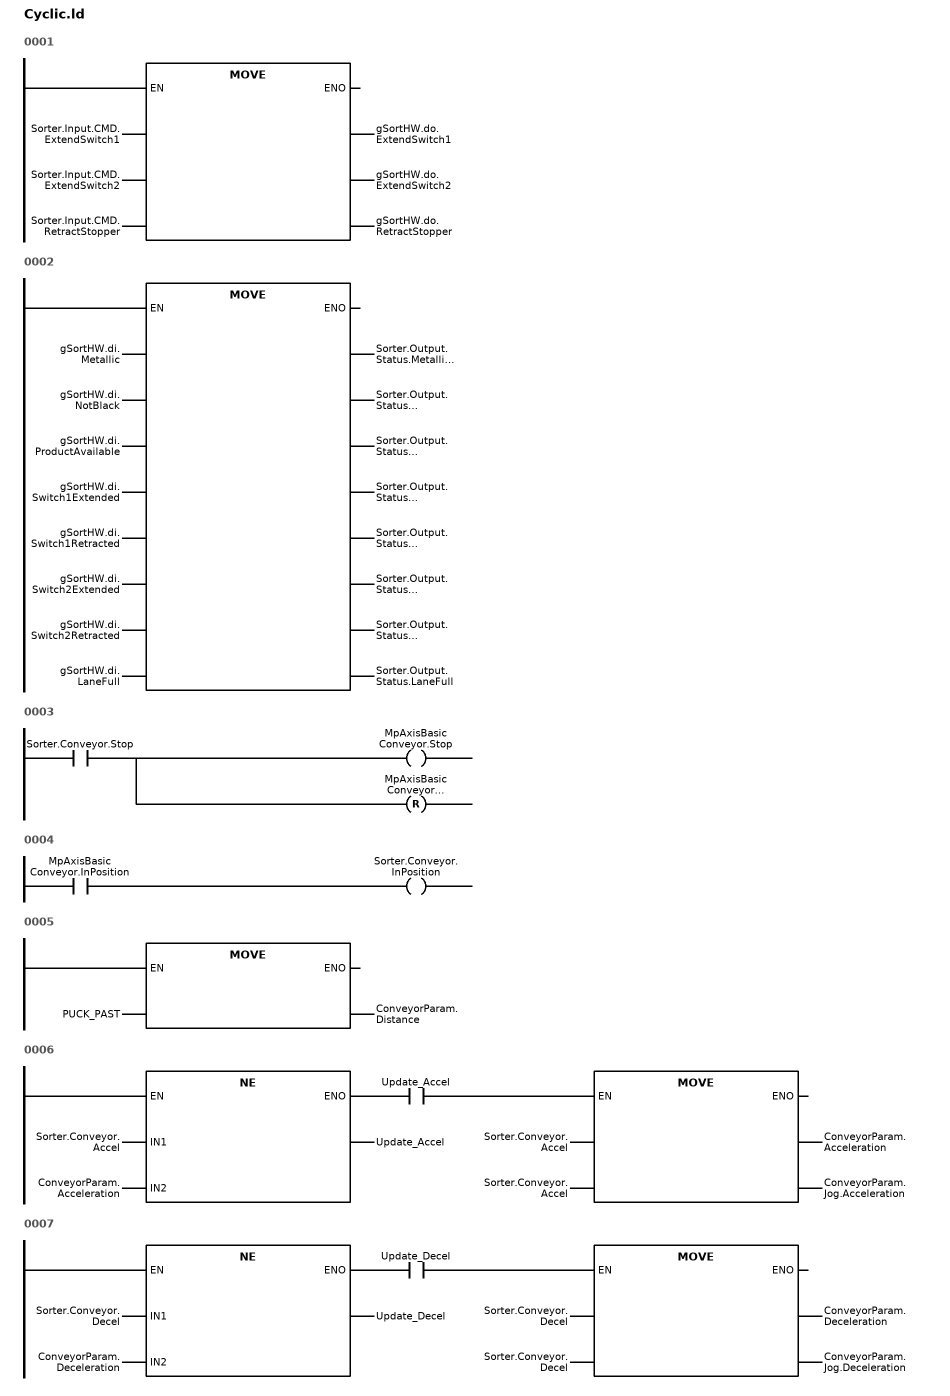
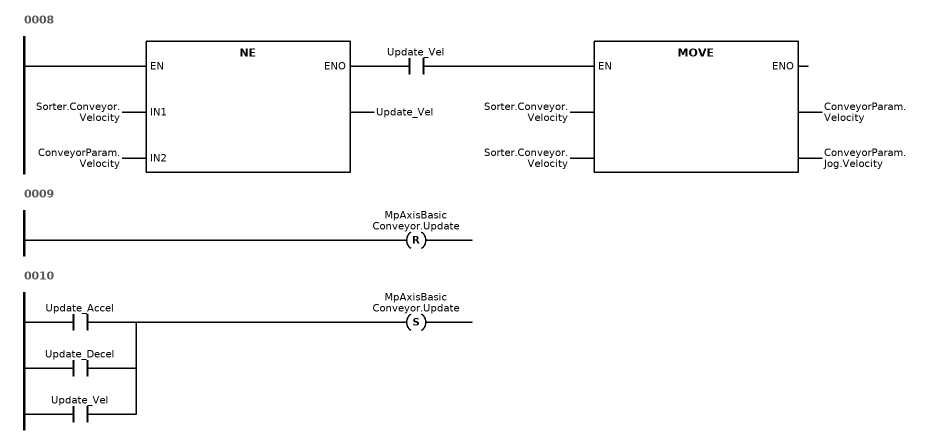
Ladder, written as Structured Text:
```iecst
(*********************************************************************************
 * Copyright:
 * Author:
 * Created:   	March 8, 2019/12:42 PM
 * Description:
 *********************************************************************************)
PROGRAM _CYCLIC
(* Network 1 *)
gSortHW.do.ExtendSwitch1 := Sorter.Input.CMD.ExtendSwitch1;
gSortHW.do.ExtendSwitch2 := Sorter.Input.CMD.ExtendSwitch2;
gSortHW.do.RetractStopper := Sorter.Input.CMD.RetractStopper;

(* Network 2 *)
Sorter.Output.Status.MetallicProduct := gSortHW.di.Metallic;
Sorter.Output.Status.ProductNotBlack := gSortHW.di.NotBlack;
Sorter.Output.Status.ProductAvailable := gSortHW.di.ProductAvailable;
Sorter.Output.Status.Switch1Extended := gSortHW.di.Switch1Extended;
Sorter.Output.Status.Switch1Retracted := gSortHW.di.Switch1Retracted;
Sorter.Output.Status.Switch2Extended := gSortHW.di.Switch2Extended;
Sorter.Output.Status.Switch2Retracted := gSortHW.di.Switch2Retracted;
Sorter.Output.Status.LaneFull := gSortHW.di.LaneFull;

(* Network 3 *)
MpAxisBasicConveyor.Stop := Sorter.Conveyor.Stop;
IF Sorter.Conveyor.Stop THEN MpAxisBasicConveyor.MoveVelocity := FALSE; END_IF;

(* Network 4 *)
Sorter.Conveyor.InPosition := MpAxisBasicConveyor.InPosition;

(* Network 5 *)
ConveyorParam.Distance := PUCK_PAST;

(* Network 6 *)
Update_Accel := Sorter.Conveyor.Accel <> ConveyorParam.Acceleration;
IF Update_Accel THEN
    ConveyorParam.Acceleration := Sorter.Conveyor.Accel;
    ConveyorParam.Jog.Acceleration := Sorter.Conveyor.Accel;
END_IF;

(* Network 7 *)
Update_Decel := Sorter.Conveyor.Decel <> ConveyorParam.Deceleration;
IF Update_Decel THEN
    ConveyorParam.Deceleration := Sorter.Conveyor.Decel;
    ConveyorParam.Jog.Deceleration := Sorter.Conveyor.Decel;
END_IF;

(* Network 8 *)
Update_Vel := Sorter.Conveyor.Velocity <> ConveyorParam.Velocity;
IF Update_Vel THEN
    ConveyorParam.Velocity := Sorter.Conveyor.Velocity;
    ConveyorParam.Jog.Velocity := Sorter.Conveyor.Velocity;
END_IF;

(* Network 9 *)
MpAxisBasicConveyor.Update := FALSE;

(* Network 10 *)
IF Update_Accel OR Update_Decel OR Update_Vel THEN MpAxisBasicConveyor.Update := TRUE; END_IF;
END_PROGRAM
```
